   //-step-800---level--0-------------------------------------------------------------                                                 
   //            RE: crystal cool down without Ar
   //---------------------------------------------------------------------------------                                                 
           800 :                                                     
               IF #next_step[0] = #active_step[0] THEN                       
                   "APC".TI[0]       := 0;                     
                   "APC".OP_MSG      := "OP_MSG".RE_WAIT_TILL_XT_COOL;
                   "LT".AUTO_OP_CALL := FALSE;
                END_IF;

               // calculate all setpoints for this step
               // -------------------------------------                                      
               "AM_PAR_FNC_RE"();

               //argon inlet 
               //-----------
               "DC".V5_OP    := FALSE;   //close valve V5
               "DC".V6_OP    := TRUE;    //open valve V6

               //stop crystal rotation
               //---------------------
               IF ("DC".XT_ROT_CW OR "DC".XT_ROT_CCW) THEN 
                   IF "SysTick1s" THEN
                       "AC".SET_XT_ROT := "AC".SET_XT_ROT - ("CNF".RE_RMP_RTE_XT_ROT / 60.0);
                   END_IF;
               END_IF;

               IF ("AC".SET_XT_ROT <= 1.0)  THEN
                   "AC".SET_XT_ROT   :=  0.0;
                   "DC".XT_ROT_CW    :=  FALSE;
                   "DC".XT_ROT_CCW   :=  FALSE;
               END_IF;

               // time till end of this step
               // --------------------------
               "APC".ACT_TME_STE := (REAL_TO_INT("PAR_MAIN".RC_XT_COOL_DN_TME) * 60) - "APC".TI[0];

               //check end condition
               //-------------------
               IF (("APC".TI[0] > (REAL_TO_INT("PAR_MAIN".RC_XT_COOL_DN_TME) * 60)) AND ("AC".SET_XT_ROT = 0.0)) THEN    
                   #end_of_step[0] := true;                            
               END_IF;

               #next_step[0] := 900; 

   //-step-900---level--0-------------------------------------------------------------                                                 
   //            RE: increase pressure in gate chamber
   //---------------------------------------------------------------------------------                                                 
           900 :                                                     
               IF #next_step[0] = #active_step[0] THEN
                   "APC".OP_MSG := "OP_MSG".VENTING_GATE;
               END_IF;

               // calculate all setpoints for this step
               // -------------------------------------                                      
               "AM_PAR_FNC_RE"();

               //vent gate chamber
               //-----------------
               IF  ("LT".V7_CLOSE AND NOT "LT".V7_OPEN)  THEN  // gate valve V7 closed ?
                   "DC".V4_OP            := TRUE;
                   "FLT".GATE_V_NOT_CLD  := FALSE;
               ELSE
                   "DC".V4_OP            := FALSE;
                   "FLT".GATE_V_NOT_CLD  := TRUE;
               END_IF;

               //check end condition
               //-------------------
               IF "DV".APS_GCH_DELAYED THEN    
                   "DC".V4_OP        := FALSE;
                   #end_of_step[0]  := true;                            
               END_IF;

               #next_step[0] := 1000; 

   //-step-1000---level--0------------------------------------------------------------                                                 
   //            RE: crystal cool down with Ar and raise crucible to start position
   //---------------------------------------------------------------------------------                                                 
          1000 :                                                     
               IF #next_step[0] = #active_step[0] THEN                       
                   "APC".TI[0]   := 0;                     
                   "APC".OP_MSG  := "OP_MSG".RE_WAIT_TILL_XT_COOL;
                END_IF;

               // calculate all setpoints for this step
               // -------------------------------------                                      
               "AM_PAR_FNC_RE"();

               // time till end of this step
               // --------------------------
               "APC".ACT_TME_STE := (REAL_TO_INT("PAR_MAIN".RC_XT_COOL_DN_TME_AR) * 60) - "APC".TI[0];

               //raise crucible to start position
               //--------------------------------
               IF ("AV".ACT_CR_POS < #cr_start_pos) THEN
                   "DC".CR_LFT_UP    :=  TRUE;    
                   "AC".SET_CR_SPD   :=  "CNF".RE_CR_SPD;
               ELSE
                   IF NOT "APC".AUTOMATIC THEN                       //stop crucible lift if puller running in manual mode
                       IF "DC".CR_LFT_UP THEN
                           "KYD".CR_LFT_OFF  :=  TRUE;
                           #cr_lft_man_off  :=  true;
                       ELSIF #cr_lft_man_off THEN 
                           "KYD".CR_LFT_OFF  :=  FALSE;
                           #cr_lft_man_off  :=  false;
                       END_IF;
                   END_IF;
                   "DC".CR_LFT_UP    :=  FALSE;    
                   "AC".SET_CR_SPD   :=  0.0;
               END_IF;

               //check end condition
               //-------------------
               IF (("APC".TI[0] > (REAL_TO_INT("PAR_MAIN".RC_XT_COOL_DN_TME_AR) * 60)) AND NOT "DC".CR_LFT_UP) THEN    
                   #end_of_step[0] := true;                            
               END_IF;

               #next_step[0] := 1050; 

   //-step-1050--level--0---------------------------------------------------------------------------------------------                                                
   //            RE: check if gate chamber is at atmospheric pressure
   //-----------------------------------------------------------------------------------------------------------------                                   
           1050 :                                                     
               IF #next_step[0] = #active_step[0] THEN                       
                   "APC".TI[0]   := 0;                     
               END_IF;

               // calculate all setpoints for this step
               // -------------------------------------                                      
               "AM_PAR_FNC_RE"();

               //check end condition
               //-------------------
               IF "DV".APS_GCH_DELAYED THEN    
                   "DC".V4_OP            := FALSE;
                   "FLT".GATE_V_NOT_CLD  := FALSE;
               ELSE
                   IF  ("LT".V7_CLOSE AND NOT "LT".V7_OPEN) THEN  // gate valve V7 closed ?
                       "DC".V4_OP            := TRUE;
                       "FLT".GATE_V_NOT_CLD  := FALSE;
                   ELSE
                       "DC".V4_OP            := FALSE;
                       "FLT".GATE_V_NOT_CLD  := TRUE;
                   END_IF;
               END_IF;

               //check end condition
               //-------------------
               IF (NOT "DC".V4_OP AND NOT "PDO".V4) THEN    
                   #end_of_step[0]  := true;                            
               END_IF;

               #next_step[0] := 1100; 

   //-step-1100--level--0---------------------------------------------------------------------------------------------                                                
   //            RE: message "remove crystal" and wait till crystal is removed  - increase crucible rot to start value
   //-----------------------------------------------------------------------------------------------------------------                                   
           1100 :                                                     
               IF #next_step[0] = #active_step[0] THEN                       
                   "APC".OP_MSG          :=  "OP_MSG".RE_REMOVE_CRYSTAL;
                   "LT".AUTO_OP_CALL     :=  TRUE;
                   "APC".TI[0]           :=  0;
                   #xt_removed          :=  false;
                   "KYD".CR_LFT_OFF      :=  FALSE;
                   "DV".MAN_ACKN_XT_RMV  :=  FALSE;
                   "LT".SHOW_XT_RMV_BTN  :=  TRUE;
               END_IF;

               // calculate all setpoints for this step
               // -------------------------------------                                      
               "AM_PAR_FNC_RE"();

               //crucible rotation set point ramp
               //--------------------------------
               IF ("SysTick1s" AND ("AC".SET_CR_ROT < #cr_start_rot)) THEN 
                   "AC".SET_CR_ROT := "AC".SET_CR_ROT + ("CNF".RE_RMP_RTE_CR_ROT / 60.0);
               END_IF;

               //built crystal removed flag
               //--------------------------
               IF NOT "PDI".LS_GCH_DOOR_CL AND "PDI".LS_GCH_DOOR_OP AND "PDI".LS_XT_HDL_SW_LOCK AND "PDI".LS_XT_SLID_FW AND "PDI".LS_UP_XT_CLP_CL THEN
                   #xt_removed := true;
               END_IF;

               //check end condition - crystal removed and puller closed again
               //-------------------------------------------------------------
               IF ("PDI".LS_GCH_DOOR_CL AND NOT "PDI".LS_GCH_DOOR_OP AND #xt_removed) OR "DV".MAN_ACKN_XT_RMV THEN 
                   //delay next step 5 seconds
                   //-------------------------
                   IF ("APC".TI[0] > 5) THEN    
                       IF ("AC".SET_CR_ROT >= #cr_start_rot) THEN  //crucible rot set point reached
                           #end_of_step[0] := true; 
                       END_IF;
                   END_IF;
               ELSE
                   "APC".TI[0] := 0;
               END_IF;

               #next_step[0] := 1200; 

   //-step-1200--level--0--------------------------------------------------------------                                                 
   //            RE: pump down gate chamber
   //----------------------------------------------------------------------------------                                                 
          1200 :                                                     
               IF #next_step[0] = #active_step[0] THEN
                   "APC".OP_MSG          := "OP_MSG".PUMP_DOWN_GATE;     
                   "LT".AUTO_OP_CALL     := FALSE;
                   "LT".SHOW_XT_RMV_BTN  := FALSE;
               END_IF;

               // calculate all setpoints 
               // -----------------------
               "AM_PAR_FNC_RE" ();

               //start vacuum pump
               //-----------------
               "DC".P3_ON := TRUE;

               //check if final pressure is reached
               //----------------------------------
               IF ("AV".ACT_PRS_GCH <= "PAR_MAIN".RC_PRG_STR_PRS)  THEN
                   "DC".V3_OP    := FALSE;  //close vacuum valve to gate chamber

               ELSE
                   "DC".V3_OP    := TRUE;   //open vacuum valve to gate chamber

               END_IF;

               //check end condition
               //-------------------
               IF NOT "PDO".V3 AND NOT "DC".V3_OP THEN     //vacuum valve V3 closed?
                   #end_of_step[0] := true;                            
               END_IF;

               #next_step[0] := 1300; 

   //-step-1300---level--0------------------------------------------------------------                                                 
   //            RE: purge Ar to furnace
   //---------------------------------------------------------------------------------                                                 
          1300 :                                                     
               IF #next_step[0] = #active_step[0] THEN
                   "APC".OP_MSG  := "OP_MSG".VENTING_GATE;       
                   "APC".TI[0]   :=  0;                                           
               END_IF;

               // calculate all setpoints 
               // -----------------------
               "AM_PAR_FNC_RE" ();

               // time till end of this step
               // --------------------------
               "APC".ACT_TME_STE := REAL_TO_INT("PAR_MAIN".RC_PRG_TME) - "APC".TI[0];

               //start purging
               //-------------
               IF (("APC".TI[0] <= REAL_TO_INT("PAR_MAIN".RC_PRG_TME)) AND NOT "PDI".GCH_APS)  THEN 
                   IF  ("LT".V7_CLOSE AND NOT "LT".V7_OPEN)THEN  // gate valve V7 closed ?
                       "DC".V4_OP            := TRUE;
                       "FLT".GATE_V_NOT_CLD  := FALSE;
                   ELSE
                       "DC".V4_OP            := FALSE;
                       "FLT".GATE_V_NOT_CLD  := TRUE;
                       "APC".TI[0]           := 0;
                   END_IF;
               //purging over
               //------------
               ELSE 
                   "DC".V4_OP            := FALSE;
                   "FLT".GATE_V_NOT_CLD  := FALSE;
                   #end_of_step[0]      := true;                            
               END_IF;

               #next_step[0] := 1400;   

   //-step-1400---level--0------------------------------------------------------------                                                 
   //            RE: check if additional purge cycle is requested
   //---------------------------------------------------------------------------------                                                 
          1400 :                                                     
               IF #next_step[0] = #active_step[0] THEN
                   "APC".OP_MSG  :=  "OP_MSG".BLANK;       
                   "APC".TI[0]   :=  0;            
                   #prg_cyc_cnt :=  #prg_cyc_cnt + 1;    //count amount of purge cycles                              
               END_IF;

               //delay switching to next step
               //----------------------------
               IF ("APC".TI[0] > 2) THEN
                   #end_of_step[0] := true;                            
               END_IF;

               //select next step
               //----------------
               IF (#prg_cyc_cnt >= REAL_TO_INT("PAR_MAIN".RC_AMT_PRG_CYC)) THEN
                   #next_step[0] := 1500; 
               ELSE
                   #next_step[0] := 1200; 
               END_IF;

   //-step-1500--level--0-------------------------------------------------------------                                                 
   //            RE: pump down gate chamber
   //---------------------------------------------------------------------------------                                                 
           1500 :                                                     
               IF #next_step[0] = #active_step[0] THEN                       
                   "APC".OP_MSG := "OP_MSG".PUMP_DOWN_GATE;
               END_IF;

               // calculate all setpoints for this step
               // -------------------------------------                                      
               "AM_PAR_FNC_RE"();

               //open vacuum valve to gate chamber
               //---------------------------------
               "DC".V3_OP    := TRUE;   

               //check end condition
               //-------------------
               IF ("AV".ACT_PRS_GCH < ("PAR_MAIN".RC_FIN_PRS_PMP_DN / 1000.0)) THEN        //unit of pressure is 10^-3 mbar
                   #end_of_step[0] := true;                            
               END_IF;

               #next_step[0] := 1600; 

   //-step-1600--level--0-------------------------------------------------------------                                                 
   //            RE: fill gate chamber with Argon
   //---------------------------------------------------------------------------------                                                 
           1600 :                                                     
               IF #next_step[0] = #active_step[0] THEN                       
                   "APC".OP_MSG := "OP_MSG".VENTING_GATE;
               END_IF;

               // calculate all setpoints for this step
               // -------------------------------------                                      
               "AM_PAR_FNC_RE"();

               //close vacuum valve to gate chamber
               //----------------------------------
               "DC".V3_OP    := FALSE;   

               //check end condition
               //-------------------
               IF (("AV".ACT_PRS_GCH - "CNF".RE_PRS_DIFF) < "AV".ACT_PRS_FCH) THEN    
                   IF  ("LT".V7_CLOSE AND NOT "LT".V7_OPEN) THEN  // gate valve V7 closed ?
                       "DC".V4_OP            := TRUE;
                       "FLT".GATE_V_NOT_CLD  := FALSE;
                   ELSE
                       "DC".V4_OP            := FALSE;
                       "FLT".GATE_V_NOT_CLD  := TRUE;
                   END_IF;
               ELSE      
                   "DC".V4_OP            := FALSE;
                   "FLT".GATE_V_NOT_CLD  := FALSE;
                   #end_of_step[0]      := true;                            
               END_IF;

               #next_step[0] := 1700; 

   //-step-1700--level--0-------------------------------------------------------------                                                 
   //            RE: message "open gate valve"
   //---------------------------------------------------------------------------------                                                 
           1700:                                                     
               IF #next_step[0] = #active_step[0] THEN                       
                   "APC".OP_MSG      := "OP_MSG".OPEN_GATE_VALVE;
                   "LT".AUTO_OP_CALL := TRUE;
               END_IF;

               // calculate all setpoints for this step
               // -------------------------------------                                      
               "AM_PAR_FNC_RE"();

               //switch off auxilliary pump
               //--------------------------
               "DC".P3_ON    :=  FALSE;  

               //open V5 when gate valve not closed
               //----------------------------------
               IF (NOT "LT".V7_CLOSE) THEN
                   "DC".V5_OP := TRUE;
               END_IF;

               //DC.V7_UP     := NOT PDI.LS_V7_UP;
               //DC.V7_SW_OUT := DV.LS_V7_UP_DLY AND NOT PDI.LS_V7_SW_OUT;

               //check end condition
               //-------------------
               IF (NOT "LT".V7_CLOSE AND "LT".V7_OPEN AND "DV".LS_V7_SW_OUT_DLY) THEN   //V7 open ?
                   "DC".V6_OP            := FALSE;               //close V6   
                   #end_of_step[0]      := true;                            
               END_IF;

               #next_step[0] := 1800; 

   //-step-1800--level--0-------------------------------------------------------------                                                 
   //            RE: wait for dipping (manual triggering of further action is necessary)
   //---------------------------------------------------------------------------------                                                 
           1800:                                                     
               "APC".OP_MSG      := "OP_MSG".RE_WAIT_FOR_DIP;
               "LT".AUTO_OP_CALL := FALSE;

               // calculate all setpoints for this step
               // -------------------------------------                                      
               "AM_PAR_FNC_RE"();

               #next_step[0] := 1800;                               // E N D

       END_CASE;

       #start_previous := #start;                                    //save start input for next call 
       #cont_previous := "APC".CONT;                                  //save cont input for next call 
       #resume_previous := "APC".RESUME;                              //save resume input for next call
       #jump_previous := "APC".JUMP;                                  //save jump input for next call
       #single_previous := "APC".SINGLE;                              //save single input for next call
END_FUNCTION_BLOCK

FUNCTION_BLOCK "AM_EMG"   // FB205, SCL
{ S7_Optimized_Access := 'FALSE' }
VERSION : 0.0
// --------------------------------------------------------------------------------
//     program     :    AM_EMG
//     description :    apc emergency module  
//     name        :    G. Eibelsh鋟ser
//     date        :    02.11.2004
// 
//     revision    :    
//     name        :    
//     date        :    
//                     (c)CGS
//     --------------------------------------------------------------------------------
   VAR_INPUT
      start : Bool;   // start sequence, activate step 10 (impulse triggered)
   END_VAR
   VAR
      start_previous : Bool;   // start input value of last call
      cont_previous : Bool;   // cont input value of last call
      resume_previous : Bool;   // resume input value of last call
      jump_previous : Bool;   // jump input value of last call
      single_previous : Bool;   // single input value of last call
      active_step : Array[0..7] of Int;   // active step number for sequence level 0..7
      next_step : Array[0..7] of Int;   // next step number for sequence level 0..7
      hold_step : Array[0..7] of Int;   // step number of step on hold
      end_of_step : Array[0..7] of Bool;   // active step is done flag for sequence 0..7
      EndOfStep : Bool;   // default value for active step is done flag
      cont_enable : Array[0..7] of Bool;   // enable continue function
      ContEnable : Bool;   // default value for enable continue function
      cr_in_pos : Bool;   // crucible in safe position
      xt_in_pos : Bool;   // crystal in safe position
      set_xt_pos : Real;   // setpoint crystal position
      set_cr_pos : Real;   // setpoint crucible position
      start_pos_xt : Real;
   END_VAR
BEGIN


       "APC".STATUS := "APC".EMG;                                      // set apc status               

       "AM_SEQUENCE_CTL" (start_p            := #start,               // control sequence
                        start_previous_p   := #start_previous,
                        cont_previous_p    := #cont_previous, 
                        resume_previous_p  := #resume_previous,
                        jump_previous_p    := #jump_previous,
                        single_previous_p  := #single_previous,
                        active_step_p      := #active_step, 
                        next_step_p        := #next_step,
                        hold_step_p        := #hold_step, 
                        end_of_step_p      := #end_of_step, 
                        cont_enable_p      := #cont_enable); 


       CASE #active_step[0] OF    //sequence level_0
   //step--0-----level--0-------------------------------------------------off--(sequence off)--------------
           0    :                                                  
                #next_step[0] := 0;

   //step--1-----level--0-------------------------------------------------hold-(test sequence)-------------
           1   :                                                       
               IF #next_step[0] = #active_step[0] THEN                   //init step     
                   //init code
                   ; 
               END_IF;
               //step code                                             //do step
               ;
   //-step-10----level--0----------------------------------------------main-(start sequence)---------------                                                 
   //-step-10----level--0-------------------------------------------------------------                                                 
   //            EMG: init emergency sequence
   //---------------------------------------------------------------------------------                                                 
           10  :  

               // enable automatic mode
               // ---------------------
               "DC".MOD_AUT_ENB  := TRUE;

               "DV".HOR_OPP  := FALSE;
               "DV".LMP_OR   := TRUE;

               #cr_in_pos   := FALSE;
               #xt_in_pos   := FALSE;

               // init rotation drives
               // --------------------
               "DC".XT_ROT_CW    := FALSE;       
               "DC".XT_ROT_CCW   := FALSE;     

               "DC".CR_ROT_CW    := FALSE;    
               "DC".CR_ROT_CCW   := FALSE;   

               "AC".SET_XT_SPD   := 0.0;
               "AC".SET_XT_ROT   := 0.0;
               "AC".SET_CR_SPD   := 0.0;
               "AC".SET_CR_ROT   := 0.0;

               // heater
               // ------
               "DC".HTR_1_ON     :=  FALSE;                    
               "DC".HTR_2_ON     :=  FALSE;

               //mobile feeder
               //-------------
               "DC".MOB_FDR_MVE_IN_SEQ_ON    :=  FALSE;
               IF ("LT".MOB_FDR_DCK_DONE AND ("DV".FDG_MVE_IN_SEQ_DONE OR NOT "DV".FDG_MVE_OUT_SEQ_DONE)) THEN 
                   "DC".MOB_FDR_MVE_OUT_SEQ_ON   :=  TRUE;
               ELSE
                   "DC".MOB_FDR_MVE_OUT_SEQ_ON   :=  FALSE;
               END_IF;

               "DC".MOB_FDR_VIB_ON           :=  FALSE;
               "FLT".MOB_FDR_NOT_DCK         :=  FALSE;
               "FLT".MOB_FDR_STP_PARA        :=  FALSE;

               // init measurement system
               // -----------------------
               "DC".CAM_ISP_ON   :=  FALSE;          //inspection off
               "DC".CAM_INIT     :=  FALSE;
               "DC".CAM_MLT      :=  FALSE;
               "DC".CAM_DIP      :=  FALSE;
               "DC".CAM_DIA      :=  TRUE;
               "DC".CAM_SEL_1    :=  TRUE;
               "DC".CAM_SEL_2    :=  FALSE;

               // control loops
               // -------------
               "DC".CTL_DIA_ON       := FALSE;              // all control loops off
               "DC".CTL_GRW_RTE_ON   := FALSE;
               "DC".CTL_PULL_RTE_ON  := FALSE;
               "DC".CTL_CRUC_ROT_ON  := FALSE;
               "DC".CTL_MLT_LVL_ON   := FALSE;
               "DC".CTL_MLT_1_TMP_ON := FALSE;
               "DC".CTL_MLT_2_TMP_ON := FALSE;
               "DC".CTL_MLT_DRIFT_ON := FALSE;
               "DC".CTL_GAP_ON       := FALSE;

               "DC".CTL_HTR_1_TMP_ON := FALSE;             // heater temp loop on
               "DC".CTL_HTR_2_TMP_ON := FALSE;

               "DC".CTL_PRS_ON        := TRUE;            // pressure control on

               "DC".CTL_SI_FDR_ON    := FALSE;
               "DC".CTL_DOP_FDR_ON   := FALSE;

               #end_of_step[0]  :=  true;
               #next_step[0] := 100;

   //-step-100---level--0-------------------------------------------------------------                                                 
   //            EMG: set control immediately to automatic mode
   //---------------------------------------------------------------------------------                                                 
           100 :                                                     

               "APC".AUTOMATIC       :=  TRUE;               
               "APC".ACT_TME_PROC    :=  0;          //reset phase time
               "APC".ACT_TME_STE     :=  0;          // reset time of step

               "APC".OP_MSG := "OP_MSG".BLANK;

               #end_of_step[0]  :=  true;                            
               #next_step[0]    :=  200;

   //-step-200---level--0-------------------------------------------------------------                                                 
   //            EMG: positioning of crystal and crucible
   //---------------------------------------------------------------------------------                                                 
           200 :   

               IF #next_step[0] = #active_step[0] THEN
                   //reset initial temperature and power setpoints
                   //----------------------------------------------
                   "DIS".HTR_1_TMP_SET_PHA_STR   :=  0.0;
                   "DIS".HTR_2_PWR_SET_PHA_STR   :=  0.0;

                   #start_pos_xt    :=  "AV".ACT_XT_POS;      //store actual crystal position                                                
               END_IF;

               //check limits of crucible movement
               //---------------------------------
               IF ("PAR_MAIN".MCONST_EMG_CR_POS < "PAR_MAIN".MCONST_LIM_CR_DN) THEN
                   #set_cr_pos := "PAR_MAIN".MCONST_LIM_CR_DN;
               ELSIF ("PAR_MAIN".MCONST_EMG_CR_POS > "PAR_MAIN".MCONST_LIM_CR_UP)  THEN
                   #set_cr_pos := "PAR_MAIN".MCONST_LIM_CR_UP;
               ELSE
                   #set_cr_pos := "PAR_MAIN".MCONST_EMG_CR_POS;       //set target position of crubible lift
               END_IF;

               "DC".CR_LFT_FST := TRUE;  //activate crucible fast flag

               //call crucible positioning module
               //--------------------------------
               "AM_CR_DRV_MOVE_DB"(set_pos   := #set_cr_pos,
                                               set_spd := "PAR_MAIN".MCONST_EMG_CR_SPD,
                                               act_pos := "AV".ACT_CR_POS, 
                                               cnf     := "CNF".CNF_CR_POS, 
                                               out_up  := "DC".CR_LFT_UP,
                                               out_dn  := "DC".CR_LFT_DN, 
                                               out_spd := "AC".SET_CR_SPD,
                                               done    := #cr_in_pos);

               //check upper limit of crystal movement
               //-------------------------------------
               IF ((#start_pos_xt - "PAR_MAIN".MCONST_EMG_XT_LFT_DIST) < "PAR_MAIN".MCONST_LIM_XTAL_UP) THEN
                   #set_xt_pos := "PAR_MAIN".MCONST_LIM_XTAL_UP;
               ELSE
                   #set_xt_pos := #start_pos_xt - "PAR_MAIN".MCONST_EMG_XT_LFT_DIST; //calculate target position crystal lift
               END_IF;

               //do lifting up of crystal
               //------------------------
               IF ("AV".ACT_XT_POS > #set_xt_pos) THEN
                   "DC".XT_LFT_UP    :=  TRUE;
                   "AC".SET_XT_SPD   :=  "PAR_MAIN".MCONST_EMG_XT_SPD;

                   IF ("AC".SET_XT_SPD > "CNF_XT_LFT_LZ950".MAX_SPEED)   THEN
                       "DC".XT_LFT_FST := TRUE;       
                   ELSE
                       "DC".XT_LFT_FST := FALSE;
                   END_IF;

               ELSE                            //stop drive, target position reached
                   "DC".XT_LFT_UP    :=  FALSE;
                   "DC".XT_LFT_FST   :=  FALSE;       
                   "AC".SET_XT_SPD   :=  0.0;           
                   #xt_in_pos       :=  true;
               END_IF;

               //check end condition
               //-------------------
               IF #cr_in_pos AND #xt_in_pos THEN
                   #end_of_step[0]  :=  true;
               END_IF;

               #next_step[0] := 300; 

   //-step-300---level--0-------------------------------------------------------------                                                 
   //            EMG: switch to manual and wait
   //---------------------------------------------------------------------------------                                                 
           300 : 

               // disable automatic mode
               // ----------------------
               "DC".MOD_AUT_ENB  := false;

               #next_step[0] := 300;

   //---------------------------------------------------------------------------------                                                 
       END_CASE;

       #start_previous  := #start;           //save start input for next call 
       #cont_previous   := "APC".CONT;        //save cont input for next call 
       #resume_previous := "APC".RESUME;      //save resume input for next call
       #jump_previous   := "APC".JUMP;        //save jump input for next call
       #single_previous := "APC".SINGLE;      //save single input for next call
END_FUNCTION_BLOCK

FUNCTION_BLOCK "AM_BY2_RP_CALC_INC"   // FB251, SCL
{ S7_Optimized_Access := 'FALSE' }
VERSION : 0.0
// --------------------------------------------------------------------------------
//     program     :    AM_BY2_RP_CALC_INC
//     description :    Calculate increment value/100ms for crystal length ramp for 2nd body
// 
//     name        :    M.Lech  
//     date        :    23.04.01
// 
//     revision    :    
//     name        :    
//     date        :    
//                     (c) CGS
//     --------------------------------------------------------------------------------
   VAR
      t : Real;   // t in sec
      INC : Real;   // INC in mm/100msec
      INC_SUM : Real;
   END_VAR
BEGIN

      IF "PAR_MAIN".BY2_RP_TME <> 0.0 THEN               //disable ramp if time = 0.0
       IF #t < "PAR_MAIN".BY2_RP_TME AND "AV".ACT_XT_LEN >= "PAR_MAIN".BY2_LEN_RP_START THEN    
           #INC := ("PAR_MAIN".BY_XT_LEN - "KYA".ACT_BDY2_LEN)/("PAR_MAIN".BY2_RP_TME*10);          // (Ltot-Lby2)/T; inc/100msec
           #INC_SUM := #INC_SUM + #INC;
           #t := #t + 0.1;                              // t+100msec     
           "APC".OP_MSG := "OP_MSG".BY2_RAMP_ACTIVE;
       ELSE    
           "APC".OP_MSG := "OP_MSG".BLANK;
       END_IF;
      END_IF;
END_FUNCTION_BLOCK

FUNCTION_BLOCK "AM_PRS_CTRL"   // FB252, SCL
{ S7_Optimized_Access := 'FALSE' }
VERSION : 0.0
// --------------------------------------------------------------------------------
//     program     :    AM_PRS_CTRL
//     description :    Controls pressure and gas flow.
// 
//                           gas flow setp > 0:    pressure control on
// 
//                                         = 0:    pressure control off
//                                                 V4 or V1 open till pressure
//                                                 setpoint reached
// 
// 
//     name        :    D.Bruess
//     date        :    19.11.99
// 
//     revision    :    
//     name        :    
//     date        :    
//                     (c) CGS
//     --------------------------------------------------------------------------------
   VAR_INPUT
      set_prs : Real;   // setpoint for pressure
      set_flw_1 : Real;   // setpoint for gas flow 1
      set_flw_2 : Real;   // setpoint for gas flow 2
      act_prs : Real;   // actual pressure
   END_VAR
   VAR_IN_OUT
      out_V4 : Bool;   // valve for venting
      out_V5 : Bool;   // valve for gas inlet
      out_prs_ctl : Bool;   // pressure control on
      out_flw_1 : Real;   // output gas flow 1
      out_flw_2 : Real;   // output gas flow 2
      out_prs : Real;   // output pressure setpoint
      out_valve_pos : Real;   // output throttle valve pos
      done : Bool;   // done flag
   END_VAR
   VAR
      req_vac : Bool;   // request flag vacuum
      req_vent : Bool;   // request flag vent
   END_VAR
BEGIN


     #out_prs := #set_prs;

     IF ((#set_flw_1 > 0.0) OR (#set_flw_2 > 0.0)) THEN
       // pressure control on (with gas flow)
       // -----------------------------------
       #out_V4 := FALSE;
       #out_V5 := TRUE;
       #out_prs_ctl := TRUE;
       #out_flw_1 := #set_flw_1;
       #out_flw_2 := #set_flw_2;
       #req_vac := FALSE;
       #req_vent := FALSE;

       #done := TRUE;
     ELSE
       // pressure control off (no gas flow)
       // ----------------------------------
       IF (#done = TRUE) THEN
         // close all valves
         // ----------------
         #out_V4 := FALSE;
         #out_V5 := FALSE;
         #out_prs_ctl := FALSE;
         #out_flw_1 := 0.0;
         #out_flw_2 := 0.0;
         #out_valve_pos := 0.0;
         #req_vac := FALSE;
         #req_vent := FALSE;
       ELSE
         IF (#set_prs < #act_prs) THEN
           // actual pressure above setpoint
           // ------------------------------
           IF (#req_vent = TRUE) THEN
             #req_vac := FALSE;                    // done
             #req_vent := FALSE;
             #done := TRUE;
           ELSE
             #req_vac := TRUE;                     // vacuum
             #req_vent := FALSE;
           END_IF;

         ELSE;
           // actual pressure below setpoint
           // ------------------------------
           IF (#req_vac = TRUE) THEN
             #req_vac := FALSE;                    // done
             #req_vent := FALSE;
             #done := TRUE;
           ELSE
             #req_vac := FALSE;                    // venting
             #req_vent := TRUE;
           END_IF;
         END_IF;

         // pressure control off
         // --------------------
         #out_prs_ctl := FALSE;

         IF (#req_vac = TRUE) THEN
           // start vaccum
           // ------------
           #out_V4 := FALSE;
           #out_V5 := FALSE;
           #out_prs_ctl := FALSE;
           #out_flw_1 := 0.0;
           #out_flw_2 := 0.0;
           #out_valve_pos := 50.0;
         ELSE
           IF (#req_vent = TRUE) THEN
             // start venting
             // -------------
             #out_V4 := TRUE;
             #out_V5 := FALSE;
             #out_prs_ctl := FALSE;
             #out_flw_1 := 0.0;
             #out_flw_2 := 0.0;
             #out_valve_pos := 0.0;
           ELSE
             // done (no request)
             // -----------------
             #out_V4 := FALSE;
             #out_V5 := FALSE;
             #out_prs_ctl := FALSE;
             #out_flw_1 := 0.0;
             #out_flw_2 := 0.0;
             #out_valve_pos := 0.0;
           END_IF;
         END_IF;
       END_IF;
     END_IF;
END_FUNCTION_BLOCK

FUNCTION_BLOCK "AM_DRV_MOVE"   // FB253, SCL
{ S7_Optimized_Access := 'FALSE' }
VERSION : 0.0
// --------------------------------------------------------------------------------
//     program     :    AM_DRV_MOVE
//     description :    Automatic positioning function (crystal and crucible).
// 
//                             set_spd        set_pos
//                         --------------------------------------------------
//                         1)     0              x        stop
//                         2)    pos             0        up with const speed
//                         3)    neg             0        dn with const speed
//                         4)    <>0            >0        move to set_pos
// 
//                      When the drive moves to set_pos then set_spd is used as 
//                      speed setpoint. If the actual position is (set_pos +- delta)
//                      then the speed setpoint is reduced. "delta" is calculated
//                      from the setpoint for the speed and from some configuration
//                      data. When the drive is in position the done flag is set.
//                      The positioning is restarted when the done flag is reset.
// 
//     name        :    D.Bruess
//     date        :    04.11.99
// 
//     revision    :    
//     name        :    
//     date        :    
//                     (c) CGS
//     --------------------------------------------------------------------------------
   VAR_INPUT
      set_pos : Real;   // setpoint for new position (0...max)
      set_spd : Real;   // setpoint for speed (0...max)
      act_pos : Real;   // actual position
      cnf : Struct
         d0 : Real;   // distance for switching to red. speed
         td : Real;   // delay time
         t_ramp : Real;   // time to reduce speed from v_max to 0
         v_max : Real;   // max speed in fast mode
         v_low : Real;   // min value for reduced speed
      END_STRUCT;
   END_VAR
   VAR_IN_OUT
      out_up : Bool;   // direction of movement = up
      out_dn : Bool;   // direction of mevement = down
      out_spd : Real;   // calculated setpoint speed
      done : Bool;   // a) set_pos=0: drive moves with const speeed
   END_VAR
   VAR
      delta : Real;   // position range for reduced setpoint
      pos_req : Bool;   // positioning has been started
   END_VAR
   VAR_TEMP
      set_spd_abs : Real;   // positive value of setpoint
      set_spd_reduced : Real;   // reduced speed setpoint
   END_VAR
BEGIN


     // calculate setpoints for speed and reduced speed
     // -----------------------------------------------
     #set_spd_abs := ABS (#set_spd);
     IF (#set_spd_abs > #cnf.v_low) THEN
       #set_spd_reduced := #cnf.v_low;
     ELSE
       #set_spd_reduced := #set_spd_abs;
     END_IF;

     // calculate distance for reduced speed
     // ------------------------------------
     #delta := #cnf.d0 +
              #cnf.td * #set_spd_abs / 60.0 +
              0.5 * #cnf.t_ramp * #set_spd_abs * #set_spd_abs / (#cnf.v_max * 60.0); 


     IF (#set_spd = 0.0) THEN
       // stop drive
       // ----------
       #out_up := FALSE;
       #out_dn := FALSE;
       #out_spd := 0.0;
       #done := TRUE;

     ELSE
       IF (#set_pos = 0.0) THEN
         // move up/dn with const speed
         // ---------------------------
         IF (#set_spd > 0.0) THEN
           // move up
           // -------
           #out_up := TRUE;
           #out_dn := FALSE;
           #out_spd := #set_spd_abs;
           #done := TRUE;

         ELSE
           // move down
           // ---------
           #out_up := FALSE;
           #out_dn := TRUE;
           #out_spd := #set_spd_abs;
           #done := TRUE;

         END_IF;

       ELSE
         IF ((#set_pos = #act_pos) OR (#done)) THEN
           // stop drive
           // ----------
           #out_up := FALSE;
           #out_dn := FALSE;
           #out_spd := 0.0;
           #done := TRUE;

         ELSE
           IF ((#act_pos < (#set_pos - #delta)) AND (#delta < #set_pos)) THEN
             // fast up
             // -------
             #out_up := TRUE;
             #out_dn := FALSE;
             #out_spd := #set_spd_abs;
             #pos_req := TRUE;

           ELSE
             IF (#act_pos > (#set_pos + #delta)) THEN
               // fast down
               // ---------
               #out_up := FALSE;
               #out_dn := TRUE;
               #out_spd := #set_spd_abs;
               #pos_req := TRUE;

             ELSE
               IF (#act_pos < #set_pos) THEN
                 IF (#pos_req AND #out_dn) THEN
                   // stop drive
                   // ----------
                   #out_up := FALSE;
                   #out_dn := FALSE;
                   #out_spd := 0.0;
                   #done := TRUE;

                 ELSE
                   // move up (with reduced speed)
                   // ----------------------------
                   #out_up := TRUE;
                   #out_dn := FALSE;
                   #out_spd := #set_spd_reduced;
                   #pos_req := TRUE;

                 END_IF;

               ELSE
                 IF (#pos_req AND #out_up) THEN
                   // stop drive
                   // ----------
                   #out_up := FALSE;
                   #out_dn := FALSE;
                   #out_spd := 0.0;
                   #done := TRUE;

                 ELSE
                   // move down (with reduced speed)
                   // ------------------------------
                   #out_up := FALSE;
                   #out_dn := TRUE;
                   #out_spd := #set_spd_reduced;
                   #pos_req := TRUE;

                 END_IF;
               END_IF;
             END_IF;
           END_IF;
         END_IF;
       END_IF;
     END_IF;


     // reset flag when positioning done
     // --------------------------------
     IF (#done = TRUE) THEN
       #pos_req := FALSE;
     END_IF;
END_FUNCTION_BLOCK

FUNCTION_BLOCK "SM_FLT_SETP_DEV_PRC"   // FB260, SCL
{ S7_Optimized_Access := 'FALSE' }
VERSION : 0.0
// --------------------------------------------------------------------------------
//     program     :    SM_CALL_FLT_SETP_DEV_PRC
//     description :    Setpoint deviation processing
//                      Call module to check deviation and set alarm flag       
//     name        :    G. Eibelsh鋟ser
//     date        :    04.02.00
// 
//     revision    :    alarms for magnet current and resistance
//     name        :    M. Lech
//     date        :    03.11.00
//     
//     revision    :    
//     name        :
//     date        :   
//                     (c) CGS
//     --------------------------------------------------------------------------------
   VAR
      ACT_FLT_TME_GAS_1_FLW : Int;   // actual fault time gas flow 1
      ACT_FLT_TME_GAS_2_FLW : Int;   // actual fault time gas flow 2
      ACT_FLT_TME_PRS : Int;   // actual fault time pressure
      ACT_FLT_TME_HTR_1_PWR : Int;   // actual fault time heater 1 power
      ACT_FLT_TME_HTR_2_PWR : Int;   // actual fault time heater 2 power
      ACT_FLT_TME_MAG_1_CUR : Int;   // actual fault time magnet 1 current
      ACT_FLT_TME_MAG_2_CUR : Int;   // actual fault time magnet 2 current
      ACT_FLT_TME_DIA_NECK_MIN : Int;   // actual fault time neck diameter below limit
      ACT_FLT_TME_XT_GRO : Int;   // actual fault time crystal growth
      ACT_FLT_TME_XT_1_DIA : Int;   // actual fault time crystal 1 diameter
      ACT_FLT_TME_XT_2_DIA : Int;   // actual fault time crystal 2 diameter
      ACT_FLT_TME_PULL_SPD_NE : Int;   // actual fault time average pull speed neck
      ACT_FLT_TME_PULL_SPD_BY1 : Int;   // actual fault time average pull speed body part 1
      ACT_FLT_TME_PULL_SPD_BY2 : Int;   // actual fault time average pull speed body part 2
   END_VAR
   VAR_TEMP
      dev_flt_gas_1_flw : Bool;   // fault flag gas flow 1
      dev_flt_gas_2_flw : Bool;   // fault flag gas flow 2
      dev_flt_prs : Bool;   // fault flag pressure
      dev_flt_htr_1_pwr : Bool;   // fault flag heater 1 power
      dev_flt_htr_2_pwr : Bool;   // fault flag heater 2 power
      dev_flt_mag_1_cur : Bool;   // fault flag magnet 1 current
      dev_flt_mag_2_cur : Bool;   // fault flag magnet 2 current
      dev_flt_dia_neck_min : Bool;   // fault flag neck diameter below limit
      dev_flt_xt_gro : Bool;   // fault flag crystal growth
      dev_flt_xt_1_dia : Bool;   // fault flag crystal diameter part 1
      dev_flt_xt_2_dia : Bool;   // fault flag crystal diameter part 2
      dev_flt_avg_pull_spd_ne : Bool;   // fault flag average pull speed neck
      dev_flt_avg_pull_spd_by1 : Bool;   // fault flag average pull speed body part 1
      dev_flt_avg_pull_spd_by2 : Bool;   // fault flag average pull speed body part 2
   END_VAR
BEGIN

       //------------------------------------     
       //fault setpoint deviation: gas flow 1
       //------------------------------------    
       "SM_FLT_SETP_DEV_DLY" (act_value        := "DIS".ACT_GAS_1_FLW,       
                            set_value        := "DIS".SET_GAS_1_FLW,
                            max_dev          := "PAR_MAIN".LIM_GAS_1_FLW,
                            delay_time       := "PAR_MAIN".LIM_GAS_FLW_DLY,
                            enable           := ("PDO".V5 OR "PDO".V6), 
                            fault            => #dev_flt_gas_1_flw);

       "FLT".GAS_FLW_1_OUT_OF_RNG := "SysOndelay"
                                   (DIN     := #dev_flt_gas_1_flw,                     // fault input
                                    SetTime := REAL_TO_INT("PAR_MAIN".LIM_GAS_FLW_DLY), // delay time
                                    ActTime := #ACT_FLT_TME_GAS_1_FLW,                 // actual time value
                                    Tick    := "SysTick1s");                            // timebase (1s)

       //------------------------------------ 
       //fault setpoint deviation: gas flow 2
       //------------------------------------    
       "SM_FLT_SETP_DEV_DLY" (act_value        := "DIS".ACT_GAS_2_FLW,       
                            set_value        := "DIS".SET_GAS_2_FLW,
                            max_dev          := "PAR_MAIN".LIM_GAS_2_FLW,
                            delay_time       := "PAR_MAIN".LIM_GAS_FLW_DLY,
                            enable           := ("PDO".V5 OR "PDO".V6),
                            fault            => #dev_flt_gas_2_flw);

       "FLT".GAS_FLW_2_OUT_OF_RNG := "SysOndelay"
                                   (DIN     := #dev_flt_gas_2_flw,                     // fault input
                                    SetTime := REAL_TO_INT("PAR_MAIN".LIM_GAS_FLW_DLY), // delay time
                                    ActTime := #ACT_FLT_TME_GAS_2_FLW,                 // actual time value
                                    Tick    := "SysTick1s");                            // timebase (1s)

       //------------------------------------ 
       //fault setpoint deviation: pressure
       //------------------------------------    
       "SM_FLT_SETP_DEV_DLY" (act_value        := "DIS".ACT_PRS_CLF,       
                            set_value        := "DIS".SET_PRS_FNC,
                            max_dev          := "PAR_MAIN".LIM_PRS,
                            delay_time       := "PAR_MAIN".LIM_GAS_FLW_DLY,
                            enable           := "LT".CTL_PRS_ON,
                            fault            => #dev_flt_prs);

       "FLT".PRS_OUT_OF_RNG := "SysOndelay"
                             (DIN     := #dev_flt_prs,                              // fault input
                              SetTime := REAL_TO_INT("PAR_MAIN".LIM_GAS_FLW_DLY),    // delay time
                              ActTime := #ACT_FLT_TME_PRS,                          // actual time value
                              Tick    := "SysTick1s");                               // timebase (1s)

       //---------------------------------------- 
       //fault setpoint deviation: heater 1 power
       //----------------------------------------    
       "SM_FLT_SETP_DEV_DLY" (act_value        := "DIS".ACT_HTR_1_PWR,       
                            set_value        := "DIS".SET_HTR_1_PWR,
                            max_dev          := "PAR_MAIN".LIM_HTR_1_PWR,
                            delay_time       := "PAR_MAIN".LIM_HTR_PWR_DLY,
                            enable           := "LT".HTR_1_ON,
                            fault            => #dev_flt_htr_1_pwr);

       "FLT".HTR_1_PWR_OUT_OF_RNG := "SysOndelay"
                                   (DIN     := #dev_flt_htr_1_pwr,                        // fault input
                                    SetTime := REAL_TO_INT("PAR_MAIN".LIM_HTR_PWR_DLY),    // delay time
                                    ActTime := #ACT_FLT_TME_HTR_1_PWR,                    // actual time value
                                    Tick    := "SysTick1s");                               // timebase (1s)

       //---------------------------------------- 
       //fault setpoint deviation: heater 2 power
       //----------------------------------------    
       "SM_FLT_SETP_DEV_DLY" (act_value        := "DIS".ACT_HTR_2_PWR,       
                            set_value        := "DIS".SET_HTR_2_PWR,
                            max_dev          := "PAR_MAIN".LIM_HTR_2_PWR,
                            delay_time       := "PAR_MAIN".LIM_HTR_PWR_DLY,
                            enable           := "LT".HTR_2_ON,
                            fault            => #dev_flt_htr_2_pwr);

       "FLT".HTR_2_PWR_OUT_OF_RNG := "SysOndelay"
                                   (DIN     := #dev_flt_htr_2_pwr,                        // fault input
                                    SetTime := REAL_TO_INT("PAR_MAIN".LIM_HTR_PWR_DLY),    // delay time
                                    ActTime := #ACT_FLT_TME_HTR_2_PWR,                    // actual time value
                                    Tick    := "SysTick1s");                               // timebase (1s)

       //---------------------------------------------
       //fault setpoint deviation: heater 1 resistance
       //---------------------------------------------   
       IF ABS("AV".ACT_HTR_1_RES_CNG) > "PAR_MAIN".LIM_HTR_1_RES    THEN
           "FLT".HTR_1_RES_OUT_OF_RNG    :=    TRUE;
       ELSE    
           "FLT".HTR_1_RES_OUT_OF_RNG    :=    FALSE;
       END_IF;

       //---------------------------------------------
       //fault setpoint deviation: heater 2 resistance
       //---------------------------------------------    
       IF ABS("AV".ACT_HTR_2_RES_CNG) > "PAR_MAIN".LIM_HTR_2_RES    THEN
           "FLT".HTR_2_RES_OUT_OF_RNG    :=    TRUE;
       ELSE    
           "FLT".HTR_2_RES_OUT_OF_RNG    :=    FALSE;
       END_IF;

       (*
       //-----------------------------------------------
       //fault setpoint deviation: magnet coil 1 current
       //-----------------------------------------------    
       SM_FLT_SETP_DEV_DLY (act_value        := DIS.ACT_MAG_1_CUR,       
                            set_value        := DIS.SET_MAG_1_CUR,
                            max_dev          := PAR_MAIN.LIM_MAG_1_CUR,
                            delay_time       := PAR_MAIN.LIM_MAG_DLY,
                            enable           := LT.MAG_ON,
                            fault            := dev_flt_mag_1_cur);

       FLT.MAG_1_CUR_OUT_OF_RNG := SysOndelay
                                   (DIN     := dev_flt_mag_1_cur,                        // fault input
                                    SetTime := REAL_TO_INT(PAR_MAIN.LIM_MAG_DLY),        // delay time
                                    ActTime := ACT_FLT_TME_MAG_1_CUR,                    // actual time value
                                    Tick    := SysTick1s);                               // timebase (1s)

       //-----------------------------------------------
       //fault setpoint deviation: magnet coil 2 current
       //-----------------------------------------------    
       SM_FLT_SETP_DEV_DLY (act_value        := DIS.ACT_MAG_2_CUR,       
                            set_value        := DIS.SET_MAG_2_CUR,
                            max_dev          := PAR_MAIN.LIM_MAG_2_CUR,
                            delay_time       := PAR_MAIN.LIM_MAG_DLY,
                            enable           := LT.MAG_ON,
                            fault            := dev_flt_mag_2_cur);

       FLT.MAG_2_CUR_OUT_OF_RNG := SysOndelay
                                   (DIN     := dev_flt_mag_2_cur,                        // fault input
                                    SetTime := REAL_TO_INT(PAR_MAIN.LIM_MAG_DLY),        // delay time
                                    ActTime := ACT_FLT_TME_MAG_2_CUR,                    // actual time value
                                    Tick    := SysTick1s);                               // timebase (1s)


       //--------------------------------------------------
       //fault setpoint deviation: magnet coil 1 resistance
       //--------------------------------------------------   
       IF ABS(AV.ACT_MAG_1_RES_CNG) > PAR_MAIN.LIM_MAG_1_RES    THEN
           FLT.MAG_1_RES_OUT_OF_RNG    :=    TRUE;
       ELSE    
           FLT.MAG_1_RES_OUT_OF_RNG    :=    FALSE;
       END_IF;


       //--------------------------------------------------
       //fault setpoint deviation: magnet coil 2 resistance
       //--------------------------------------------------   
       IF ABS(AV.ACT_MAG_2_RES_CNG) > PAR_MAIN.LIM_MAG_2_RES    THEN
           FLT.MAG_2_RES_OUT_OF_RNG    :=    TRUE;
       ELSE    
           FLT.MAG_2_RES_OUT_OF_RNG    :=    FALSE;
       END_IF;
       *)
       //------------------------------------------------------
       //fault setpoint deviation: neck diameter below limit
       //------------------------------------------------------    
       (*
       SM_FLT_SETP_DEV_DLY (act_value        := DIS.ACT_XT_DIA,       
                            set_value        := DIS.SET_XT_DIA,
                            max_dev          := PAR_MAIN.LIM_DIA_NECK_MIN,
                            delay_time       := PAR_MAIN.LIM_DIA_NECK_DLY,
                            enable           := (APC.STATUS = APC.NECK) AND DC.CTL_DIA_ON AND LT.XT_LFT_UP,
                            fault            := dev_flt_dia_neck_min);
       *)
       IF ("APC".STATUS = "APC".NECK) AND "DC".CTL_DIA_ON AND "LT".XT_LFT_UP   THEN 
           IF ("DIS".ACT_XT_DIA < "PAR_MAIN".LIM_DIA_NECK_MIN) THEN
               #dev_flt_dia_neck_min := true;
           ELSE 
               #dev_flt_dia_neck_min := false;
           END_IF;
       ELSE
           #dev_flt_dia_neck_min := false;
       END_IF;

       "FLT".NECK_DIA_BELOW_LIMIT := "SysOndelay"
                                   (DIN     := #dev_flt_dia_neck_min,                   // fault input
                                    SetTime := REAL_TO_INT("PAR_MAIN".LIM_DIA_NECK_DLY), // delay time
                                    ActTime := #ACT_FLT_TME_DIA_NECK_MIN,               // actual time value
                                    Tick    := "SysTick1s");                             // timebase (1s)

       //----------------------------------------
       //fault setpoint deviation: crystal growth
       //----------------------------------------
       "SM_FLT_SETP_DEV_DLY" (act_value        := "DIS".ACT_XTAL_GRO,       
                            set_value        := "DIS".SET_XTAL_GRO,
                            max_dev          := "PAR_MAIN".LIM_GRO,
                            delay_time       := "PAR_MAIN".LIM_GRO_DLY,
                            enable           := "DC".CTL_GRW_RTE_ON,
                            fault            => #dev_flt_xt_gro);

       "FLT".XT_GROWTH_OUT_OF_RNG := "SysOndelay"
                                   (DIN     := #dev_flt_xt_gro,                    // fault input
                                    SetTime := REAL_TO_INT("PAR_MAIN".LIM_GRO_DLY), // delay time
                                    ActTime := #ACT_FLT_TME_XT_GRO,                // actual time value
                                    Tick    := "SysTick1s");                        // timebase (1s)

       //--------------------------------------------------------
       //fault setpoint deviation: crystal diameter (body part 1)
       //--------------------------------------------------------
       IF ("APC".STATUS = "APC".BODY) AND ("DIS".ACT_XT_LEN_MM <= "PAR_MAIN".LIM_LEN_BODY1) THEN

        "SM_FLT_SETP_DEV_DLY" (act_value        := "DIS".ACT_XT_DIA,       
                             set_value        := "DIS".SET_XT_DIA,
                             max_dev          := "PAR_MAIN".LIM_DIA_BODY_1,
                             delay_time       := "PAR_MAIN".LIM_DIA_DLY,
                             enable           := "DC".CTL_DIA_ON AND "LT".XT_LFT_UP, 
                             fault            => #dev_flt_xt_1_dia);

        "FLT".XT_DIA_OUT_OF_RNG    := "SysOndelay"
                                   (DIN     := #dev_flt_xt_1_dia,                 // fault input
                                    SetTime := REAL_TO_INT("PAR_MAIN".LIM_DIA_DLY),  // delay time
                                    ActTime := #ACT_FLT_TME_XT_1_DIA,               // actual time value
                                    Tick    := "SysTick1s");                         // timebase (1s)

       //--------------------------------------------------------
       //fault setpoint deviation: crystal diameter (body part 2)
       //--------------------------------------------------------
       ELSIF ("APC".STATUS = "APC".BODY) AND ("DIS".ACT_XT_LEN_MM > "PAR_MAIN".LIM_LEN_BODY1) THEN

        "SM_FLT_SETP_DEV_DLY" (act_value        := "DIS".ACT_XT_DIA,       
                             set_value        := "DIS".SET_XT_DIA,
                             max_dev          := "PAR_MAIN".LIM_DIA_BODY_2,
                             delay_time       := "PAR_MAIN".LIM_DIA_DLY,
                             enable           := "DC".CTL_DIA_ON AND "LT".XT_LFT_UP, 
                             fault            => #dev_flt_xt_2_dia);

        "FLT".XT_DIA_OUT_OF_RNG    := "SysOndelay"
                                    (DIN     := #dev_flt_xt_2_dia,                   // fault input
                                     SetTime := REAL_TO_INT("PAR_MAIN".LIM_DIA_DLY),  // delay time
                                     ActTime := #ACT_FLT_TME_XT_2_DIA,               // actual time value
                                     Tick    := "SysTick1s");                         // timebase (1s)

       ELSE
           "FLT".XT_DIA_OUT_OF_RNG   :=  FALSE;    

       END_IF;

       //-------------------------------------------------
       //fault setpoint deviation: average pull speed neck
       //-------------------------------------------------
       IF ("APC".STATUS = "APC".NECK) THEN
        "SM_FLT_SETP_DEV_DLY" (act_value        := "DIS".ACT_XT_AV_SPD,       
                             set_value        := "DIS".SET_XT_AV_SPD,
                             max_dev          := "PAR_MAIN".LIM_AV_SPD_NE,
                             delay_time       := "PAR_MAIN".LIM_AV_SPD_DLY,
                             enable           := "DC".CTL_PULL_RTE_ON AND "LT".XT_LFT_UP,
                             fault            => #dev_flt_avg_pull_spd_ne);

        "FLT".AVG_PULL_SPD_OUT_OF_RNG:= "SysOndelay"
                                      (DIN     := #dev_flt_avg_pull_spd_ne,              // fault input
                                       SetTime := REAL_TO_INT("PAR_MAIN".LIM_AV_SPD_DLY), // delay time
                                       ActTime := #ACT_FLT_TME_PULL_SPD_NE,              // actual time value
                                       Tick    := "SysTick1s");                           // timebase (1s)

       //--------------------------------------------------------
       //fault setpoint deviation: average pull speed body part 1
       //--------------------------------------------------------
       ELSIF ("APC".STATUS = "APC".BODY) AND ("DIS".ACT_XT_LEN_MM <= "PAR_MAIN".LIM_LEN_BODY1) THEN

        "SM_FLT_SETP_DEV_DLY" (act_value       := "DIS".ACT_XT_AV_SPD,       
                            set_value        := "DIS".SET_XT_AV_SPD,
                            max_dev          := "PAR_MAIN".LIM_AV_SPD_BY1,
                            delay_time       := "PAR_MAIN".LIM_AV_SPD_DLY,
                            enable           := "DC".CTL_PULL_RTE_ON AND "LT".XT_LFT_UP,
                            fault            => #dev_flt_avg_pull_spd_by1);

         "FLT".AVG_PULL_SPD_OUT_OF_RNG:= "SysOndelay"
                                      (DIN     := #dev_flt_avg_pull_spd_by1,             // fault input
                                       SetTime := REAL_TO_INT("PAR_MAIN".LIM_AV_SPD_DLY), // delay time
                                       ActTime := #ACT_FLT_TME_PULL_SPD_BY1,             // actual time value
                                       Tick    := "SysTick1s");                           // timebase (1s)

       //--------------------------------------------------------
       //fault setpoint deviation: average pull speed body part 2
       //--------------------------------------------------------
       ELSIF ("APC".STATUS = "APC".BODY) AND ("DIS".ACT_XT_LEN_MM > "PAR_MAIN".LIM_LEN_BODY1) THEN

        "SM_FLT_SETP_DEV_DLY" (act_value        := "DIS".ACT_XT_AV_SPD,       
                             set_value        := "DIS".SET_XT_AV_SPD,
                             max_dev          := "PAR_MAIN".LIM_AV_SPD_BY2,
                             delay_time       := "PAR_MAIN".LIM_AV_SPD_DLY,
                             enable           := "DC".CTL_PULL_RTE_ON AND "LT".XT_LFT_UP,
                             fault            => #dev_flt_avg_pull_spd_by2);

        "FLT".AVG_PULL_SPD_OUT_OF_RNG:= "SysOndelay"
                                     (DIN     := #dev_flt_avg_pull_spd_by2,             // fault input
                                      SetTime := REAL_TO_INT("PAR_MAIN".LIM_AV_SPD_DLY), // delay time
                                      ActTime := #ACT_FLT_TME_PULL_SPD_BY2,             // actual time value
                                      Tick    := "SysTick1s");                           // timebase (1s)

       ELSE
           "FLT".AVG_PULL_SPD_OUT_OF_RNG :=  FALSE;

       END_IF;
END_FUNCTION_BLOCK

FUNCTION_BLOCK "BM_MCC"   // FB261, SCL
{ S7_Optimized_Access := 'FALSE' }
VERSION : 0.0
// --------------------------------------------------------------------------------
//     program     :    BM_MCC
//     description :    melt contact function block, test mode, fault setting, lights
//                          
//     name        :    G. Eibelshaeuser
//     date        :    14.02.2000
// 
//     revision    :
//     name        :
//     date        :    
//                     (c)CGS
// --------------------------------------------------------------------------------
   VAR
      mcc_enb : Bool;
      mcc_test : Bool;
      mcc_contact : Bool;
      mcc_on_tme_flag : Bool;
      mcc_off_tme_flag : Bool;
      mcc_detect_flag : Bool;
      mcc_xt_out_of_melt : Bool;
      mcc_on_tme : S5Time;
      mcc_off_tme : S5Time;
      mcc_detect : S5Time;
      mcc_flt_dly : S5Time;
   END_VAR
BEGIN


       //read peripherie input
       //---------------------
       #mcc_contact := "PDI".MCC_CONTACT_XT;

       //melt contact control enable
       //---------------------------
       IF ("APC".AUTOMATIC AND "DC".MCC_ON AND NOT #mcc_on_tme_flag) THEN
           #mcc_enb := TRUE;                                                                // mcc enable in automatic mode
       ELSIF (NOT "APC".AUTOMATIC AND ("KYD".MCC_ON  OR #mcc_enb) AND NOT "KYD".MCC_OFF) THEN     // mcc enable in manual mode
           #mcc_enb := TRUE;           
       ELSE    
           #mcc_enb := FALSE;                                                               // mcc disabled
       END_IF;

       //on time flag for melt contact control
       //-------------------------------------     
       #mcc_on_tme := S_ODT(T_NO:= "BM_MCC_ON_TME",                                           // Timer Symbol
                           S   := "DC".MCC_ON AND #mcc_detect_flag AND NOT #mcc_off_tme_flag,  // Start Condition
                           TV  := T#5s,                                                    // Time Setpoint 
                           Q   => #mcc_on_tme_flag); 

       //off time flag for melt contact control
       //--------------------------------------    
       #mcc_off_tme := S_ODT(   T_NO:= "BM_MCC_OFF_TME",                  // Timer Symbol
                               S   := #mcc_on_tme_flag AND "DC".MCC_ON,   // Start Condition
                               TV  := T#10s,                           // Time Setpoint 
                               Q   => #mcc_off_tme_flag);

       //melt contact control test mode
       //------------------------------
       IF ("APC".AUTOMATIC AND "DC".MCC_TST_ON)    THEN                                                // mcc test in automatic mode
           #mcc_test := TRUE;
       ELSIF (NOT "APC".AUTOMATIC AND ("KYD".MCC_TST_ON OR #mcc_test) AND NOT "KYD".MCC_TST_OFF)  THEN    // mcc test in manual mode
           #mcc_test := TRUE;
       ELSE    
           #mcc_test := FALSE;                                                                      // mcc test disabled
       END_IF;

       //crystal out of melt alarm
       //-------------------------
       IF (("APC".STATUS = "APC".DIPPING) OR ("APC".STATUS = "APC".REMOVAL)) THEN
           #mcc_xt_out_of_melt  := FALSE;
       ELSIF (#mcc_enb AND NOT #mcc_detect_flag) THEN
           #mcc_xt_out_of_melt  := TRUE;
       ELSE    
           #mcc_xt_out_of_melt  := FALSE;
       END_IF;

       #mcc_flt_dly := S_ODT(   T_NO:= "FLT_OUT_OF_MELT_DLY",                             // Timer Symbol
                               S   := #mcc_xt_out_of_melt AND NOT "LT".MLT_GAP_SEARCH,    // Start Condition
                               TV  := T#5s,                                            // Time Setpoint 
                               Q   => "FLT".EC_XT_OUT_OF_MELT);                          // Set alarm xtal out of melt

       //melt contact control detection flag
       //-----------------------------------
       #mcc_detect := S_OFFDT(  T_NO:= "MELT_CON_DETECT_DLY",             // Timer Symbol
                               S   := ("DC".MCC_ON AND NOT #mcc_enb) OR   // melt contact control requested, but not in check cycle
                                       #mcc_contact,                    // xtal is in melt
                               TV  :=  T#3s,                           // Time Setpoint 
                               Q   =>  #mcc_detect_flag);               // delay flag xtal in melt

       "DV".DI_MCC_CONTACT := #mcc_detect_flag;

       //set light variables on PC screen
       //--------------------------------
       "LT".MCC_ON             := #mcc_enb OR ("APC".AUTOMATIC AND "DC".MCC_ON);
       "LT".MCC_TST_ON         := #mcc_test;
       "LT".XT_MELT_CONTACT    := #mcc_detect_flag;        // 1: Melt contact, 0: No melt contact

       // write peripherie output
       //------------------------ 
       "PDO".MCC_ENB_XT  := #mcc_enb;
       "PDO".MCC_TEST_XT := #mcc_test;
END_FUNCTION_BLOCK

FUNCTION_BLOCK "BM_XT_WGT_CALC"   // FB262, SCL
{ S7_Optimized_Access := 'FALSE' }
VERSION : 0.0
// --------------------------------------------------------------------------------
//     program     :    BM_XT_WEIGHT_CALC
//     description :    calculate crystal weight in SHOULDER and BODY for 
//                      display variable     
//     name        :    G. Eibelsh鋟ser
//     date        :    22.02.2000
// 
//     revision    :    calculation after fixed pulling length change
//                      reset variable inserted
//     name        :    G. Eibelsh鋟ser
//     date        :    27.03.2006
//     
//                     (c)CGS
// --------------------------------------------------------------------------------
   VAR
      xt_pos_old : Real;
      pull_lgh_inc : Real;
      xt_wgt_inc : Real;
   END_VAR
   VAR CONSTANT
      min_pull_lgh : Real := 0.5;   // minimum pulling length between two calculation cycles in mm
   END_VAR
BEGIN


       //reset crystal weight
       //--------------------
       IF  ("APC".STATUS = "APC".PUMP_DOWN)    OR      //phase pump down active 
           ("APC".STATUS = "APC".MELTING)      OR      //phase melting active
           ("APC".STATUS = "APC".DIPPING)      OR      //phase dipping active
           ("APC".STATUS = "APC".NECK)         THEN    //phase neck active

           "AV".ACT_XT_WGT_CALC  := 0.0;
           #xt_pos_old          := "AV".ACT_XT_POS;

       //calculate crystal weight
       //------------------------
       ELSIF  ("APC".STATUS = "APC".SHOULDER) OR       //phase shoulder active
               ("APC".STATUS = "APC".BODY)     THEN    //phase body active

           //check pulling length change 
           //---------------------------
           IF ((#xt_pos_old - "AV".ACT_XT_POS) >= #min_pull_lgh) THEN

               //calculate pulling length of last calc cycle
               //-------------------------------------------
               #pull_lgh_inc    := #xt_pos_old - "AV".ACT_XT_POS;

               //store actual crystal position of this calculation cycle
               //-------------------------------------------------------
               #xt_pos_old      := "AV".ACT_XT_POS;

               //calculation of weight increment in kg
               //-------------------------------------
               #xt_wgt_inc := #pull_lgh_inc * SQR("AV".ACT_XT_DIA) * "CNF".RHO_SOL_SI_ROOM * "CNF".PI / 4;

               //calculation of weight sum in kg
               //-------------------------------
               "AV".ACT_XT_WGT_CALC := "AV".ACT_XT_WGT_CALC + #xt_wgt_inc;

           END_IF;
       END_IF;

       //display actual calculated crystal weight
       //----------------------------------------
       "DIS".ACT_XT_WGT_CALC :=  "AV".ACT_XT_WGT_CALC;
END_FUNCTION_BLOCK

FUNCTION_BLOCK "BM_OP_CALL"   // FB340, SCL
{ S7_Optimized_Access := 'FALSE' }
VERSION : 0.0
// --------------------------------------------------------------------------------
//     program     :    BM_OP_CALL
//     description :    start horn and lamp to call operator after time x
//     name        :    M.Lech
//     date        :    14.06.00
// 
//     revision    :
//     name        :
//     date        :    
//                     (c)CGS
//     --------------------------------------------------------------------------------
   VAR
      ACT_OP_CALL_TME : Int;   // actual Time
      OP_CALL_ALM : Bool;   // flag for operator call on 1Hz cycle
   END_VAR
BEGIN


       "LT".OP_CALL_ON := ("LT".OP_CALL_ON OR "KYD".OP_CALL_ON) AND NOT 
                       ("KYD".OP_CALL_OFF);

       IF "KYD".OP_CALL_ACK THEN
           #ACT_OP_CALL_TME := 0;
       END_IF;

       "LT".OP_CALL_ALM:= "SysOndelay"(DIN     := "LT".OP_CALL_ON,                    //  operator call activated
                                   SetTime := REAL_TO_INT("KYA".SET_OP_CALL_TME), // delay time
                                   ActTime := #ACT_OP_CALL_TME,                  // actual time value
                                   Tick    := "SysTick1s");                       // timebase (1s);


       IF "SysTick2s" AND  "LT".OP_CALL_ALM AND NOT #OP_CALL_ALM THEN
           #OP_CALL_ALM := TRUE;                                        //call flag on 2s cycle
       ELSIF  "SysTick200ms" AND  "LT".OP_CALL_ALM AND #OP_CALL_ALM THEN
           #OP_CALL_ALM := FALSE;
       ELSIF  NOT  "LT".OP_CALL_ALM OR NOT "LT".OP_CALL_ON   THEN       
           #OP_CALL_ALM := FALSE;
       END_IF;       

       IF "LT".OP_CALL_ALM = TRUE THEN
           "APC".OP_MSG := "OP_MSG".OP_CALL_ALM;
       END_IF;
END_FUNCTION_BLOCK

FUNCTION_BLOCK "PM_MDI"   // FB400, SCL
{ S7_Optimized_Access := 'FALSE' }
VERSION : 0.0
// --------------------------------------------------------------------------------
//     program:         PM_MDI
//     description :    automatically generated PM_MDI
//     name:            hp
//     date        :    03.02.2021
// 
//     revision:
//     name:
//     Date:
//                     (c)CGS
//     --------------------------------------------------------------------------------
   VAR
      y : Bool;
      count : Int := 8;
   END_VAR
   VAR_TEMP
      x : Bool;
   END_VAR
BEGIN


       "MDI".CB_FLT_DC24V_K2 := "PDI".CB_FLT_DC24V_K2;
       "MDI".CB_FLT_AC400V_K2 := "PDI".CB_FLT_AC400V_K2;
       "MDI".SPARE_16_2 := "PDI".SPARE_16_2;
       "MDI".CB_FLT_AC230V := "PDI".CB_FLT_AC230V;
       "MDI".SPARE_16_4 := "PDI".SPARE_16_4;
       "MDI".SPARE_16_5 := "PDI".SPARE_16_5;
       "MDI".SPARE_16_6 := "PDI".SPARE_16_6;
       "MDI".SPARE_16_7 := "PDI".SPARE_16_7;
       "MDI".SPARE_17_0 := "PDI".SPARE_17_0;
       "MDI".UPS_24V_ALM := "PDI".UPS_24V_ALM;
       "MDI".UPS_24V_NRM := "PDI".UPS_24V_NRM;
       "MDI".EMO := "PDI".EMO;
       "MDI".EMS := "PDI".EMS;
       "MDI".SPARE_17_5 := "PDI".SPARE_17_5;
       "MDI".SPARE_17_6 := "PDI".SPARE_17_6;
       "MDI".SPARE_17_7 := "PDI".SPARE_17_7;
       "MDI".P1_WRN := "PDI".P1_WRN;
       "MDI".P1_FLT := "PDI".P1_FLT;
       "MDI".P1_IS_ON := "PDI".P1_IS_ON;
       "MDI".P1_WD := "PDI".P1_WD;
       "MDI".FIL_APS := "PDI".FIL_APS;
       "MDI".MON_TMP_P2 := "PDI".MON_TMP_P2;
       "MDI".MON_TMP_P1 := "PDI".MON_TMP_P1;
       "MDI".SPARE_18_7 := "PDI".SPARE_18_7;
       "MDI".FCH_LFT_SDL_NUT := "PDI".FCH_LFT_SDL_NUT;
       "MDI".LS_FCH_LFT_DN := "PDI".LS_FCH_LFT_DN;
       "MDI".LS_FCH_HOOK_WORK := "PDI".LS_FCH_HOOK_WORK;
       "MDI".LS_FCH_HOOK_HOME := "PDI".LS_FCH_HOOK_HOME;
       "MDI".LS_TEC_FLG_DN := "PDI".LS_TEC_FLG_DN;
       "MDI".TEC_FLG_SDL_NUT := "PDI".TEC_FLG_SDL_NUT;
       "MDI".LS_V11_COV_OP := "PDI".LS_V11_COV_OP;
       "MDI".LS_V11_COV_CL := "PDI".LS_V11_COV_CL;
       "MDI".GCH_APS := "PDI".GCH_APS;
       "MDI".FCH_APS := "PDI".FCH_APS;
       "MDI".FDR_APS := "PDI".FDR_APS;
       "MDI".FIL_2_APS := "PDI".FIL_2_APS;
       "MDI".SPARE_33_4 := "PDI".SPARE_33_4;
       "MDI".SPARE_33_5 := "PDI".SPARE_33_5;
       "MDI".LS_V2_1_OP := "PDI".LS_V2_1_OP;
       "MDI".LS_V2_1_CL := "PDI".LS_V2_1_CL;
       "MDI".CB_FLT_AC400V_K5 := "PDI".CB_FLT_AC400V_K5;
       "MDI".CB_FLT_DC24V_K5 := "PDI".CB_FLT_DC24V_K5;
       "MDI".LS_MAG_LFT_UP := "PDI".LS_MAG_LFT_UP;
       "MDI".LS_MAG_LFT_DN := "PDI".LS_MAG_LFT_DN;
       "MDI".SLS_MAG_LFT := "PDI".SLS_MAG_LFT;
       "MDI".MAG_LFT_SDL_NUT1 := "PDI".MAG_LFT_SDL_NUT1;
       "MDI".MAG_LFT_SDL_NUT2 := "PDI".MAG_LFT_SDL_NUT2;
       "MDI".MAG_LFT_SDL_NUT3 := "PDI".MAG_LFT_SDL_NUT3;
       "MDI".OIL_LVL_CR_SFT := "PDI".OIL_LVL_CR_SFT;
       "MDI".LS_V1_OP := "PDI".LS_V1_OP;
       "MDI".LS_V1_CL := "PDI".LS_V1_CL;
       "MDI".MP_ENB_K5 := "PDI".MP_ENB_K5;
       "MDI".SLS_TEC_FLG_LFT := "PDI".SLS_TEC_FLG_LFT;
       "MDI".SLS_FCH_LFT := "PDI".SLS_FCH_LFT;
       "MDI".COMP_AIR_OK := "PDI".COMP_AIR_OK;
       "MDI".COMP_AIR_2_OK := "PDI".COMP_AIR_2_OK;
       "MDI".LS_V1_1_CL := "PDI".LS_V1_1_CL;
       "MDI".LS_V1_1_OP := "PDI".LS_V1_1_OP;
       "MDI".LS_V3_4_OP := "PDI".LS_V3_4_OP;
       "MDI".LS_V3_4_CL := "PDI".LS_V3_4_CL;
       "MDI".LS_V3_3_OP := "PDI".LS_V3_3_OP;
       "MDI".LS_V3_3_CL := "PDI".LS_V3_3_CL;
       "MDI".LS_V2_11_OP := "PDI".LS_V2_11_OP;
       "MDI".LS_V2_11_CL := "PDI".LS_V2_11_CL;
       "MDI".ACC_FCH_OV_PRS_1 := "PDI".ACC_FCH_OV_PRS_1;
       "MDI".ACC_FCH_OV_PRS_2 := "PDI".ACC_FCH_OV_PRS_2;
       "MDI".SPARE_48_2 := "PDI".SPARE_48_2;
       "MDI".ACC_WTR_FLW_OUT_OK := "PDI".ACC_WTR_FLW_OUT_OK;
       "MDI".ACC_WTR_FLW_IN_OK := "PDI".ACC_WTR_FLW_IN_OK;
       "MDI".ACC_WTR_TMP_OUT_OK := "PDI".ACC_WTR_TMP_OUT_OK;
       "MDI".OV_PRS_1_FLT := "PDI".OV_PRS_1_FLT;
       "MDI".OV_PRS_2_FLT := "PDI".OV_PRS_2_FLT;
       "MDI".ACC_SC_WTR_OK := "PDI".ACC_SC_WTR_OK;
       "MDI".ACC_SC_WTR_ATV := "PDI".ACC_SC_WTR_ATV;
       "MDI".ACC_SC_HTR_OK := "PDI".ACC_SC_HTR_OK;
       "MDI".ACC_SC_HTR_ATV := "PDI".ACC_SC_HTR_ATV;
       "MDI".ACC_KEY_RST := "PDI".ACC_KEY_RST;
       "MDI".ACC_CB_FLT_DC24V := "PDI".ACC_CB_FLT_DC24V;
       "MDI".ACC_UPS_24V_ALM := "PDI".ACC_UPS_24V_ALM;
       "MDI".ACC_UPS_24V_NRM := "PDI".ACC_UPS_24V_NRM;
       "MDI".DPH_RPT_DET_OK := "PDI".DPH_RPT_DET_OK;
       "MDI".ACC_CB_FLT_AC230V := "PDI".ACC_CB_FLT_AC230V;
       "MDI".SPARE_90_2 := "PDI".SPARE_90_2;
       "MDI".SPARE_90_3 := "PDI".SPARE_90_3;
       "MDI".SPARE_90_4 := "PDI".SPARE_90_4;
       "MDI".SPARE_90_5 := "PDI".SPARE_90_5;
       "MDI".SPARE_90_6 := "PDI".SPARE_90_6;
       "MDI".SPARE_90_7 := "PDI".SPARE_90_7;
       "MDI".FU_P2_RDY := "PDI".FU_P2_RDY;
       "MDI".SPARE_144_1 := "PDI".SPARE_144_1;
       "MDI".LS_GCH_UP := "PDI".LS_GCH_UP;
       "MDI".LS_GCH_DN := "PDI".LS_GCH_DN;
       "MDI".LS_GCH_SW_IN := "PDI".LS_GCH_SW_IN;
       "MDI".LS_GCH_SW_CLN := "PDI".LS_GCH_SW_CLN;
       "MDI".LS_GCH_SW_OUT := "PDI".LS_GCH_SW_OUT;
       "MDI".LS_GCH_SW_LOCK := "PDI".LS_GCH_SW_LOCK;
       "MDI".SLS_GCH_LFT := "PDI".SLS_GCH_LFT;
       "MDI".LS_TCH_UP := "PDI".LS_TCH_UP;
       "MDI".LS_TCH_DN := "PDI".LS_TCH_DN;
       "MDI".LS_TCH_SW_IN := "PDI".LS_TCH_SW_IN;
       "MDI".LS_TCH_SW_CLN := "PDI".LS_TCH_SW_CLN;
       "MDI".LS_TCH_SW_OUT := "PDI".LS_TCH_SW_OUT;
       "MDI".LS_TCH_SW_LOCK := "PDI".LS_TCH_SW_LOCK;
       "MDI".LS_TCH_TILT_0 := "PDI".LS_TCH_TILT_0;
       "MDI".LS_TCH_TILT_30 := "PDI".LS_TCH_TILT_30;
       "MDI".KEY_XT_LFT_SRV := "PDI".KEY_XT_LFT_SRV;
       "MDI".LS_V7_UP := "PDI".LS_V7_UP;
       "MDI".LS_V7_DN := "PDI".LS_V7_DN;
       "MDI".LS_V7_SW_IN := "PDI".LS_V7_SW_IN;
       "MDI".LS_V7_SW_OUT := "PDI".LS_V7_SW_OUT;
       "MDI".LS_V7_FLP_OP := "PDI".LS_V7_FLP_OP;
       "MDI".LS_V7_CLN_POS := "PDI".LS_V7_CLN_POS;
       "MDI".LS_GCH_BEL_UP := "PDI".LS_GCH_BEL_UP;
       "MDI".LS_GCH_BEL_DN := "PDI".LS_GCH_BEL_DN;
       "MDI".LS_XT_SLID_BW := "PDI".LS_XT_SLID_BW;
       "MDI".LS_XT_SLID_FW := "PDI".LS_XT_SLID_FW;
       "MDI".LS_XT_SLID_MID := "PDI".LS_XT_SLID_MID;
       "MDI".LS_XT_CLP_CON := "PDI".LS_XT_CLP_CON;
       "MDI".LS_XT_TILT_90 := "PDI".LS_XT_TILT_90;
       "MDI".LS_XT_TILT_75 := "PDI".LS_XT_TILT_75;
       "MDI".LS_UP_XT_CLP_FLT := "PDI".LS_UP_XT_CLP_FLT;
       "MDI".SPARE_275_7 := "PDI".SPARE_275_7;
       "MDI".LS_UP_XT_CLP_OP := "PDI".LS_UP_XT_CLP_OP;
       "MDI".LS_UP_XT_CLP_CL := "PDI".LS_UP_XT_CLP_CL;
       "MDI".LS_UP_XT_CLP_SAVE := "PDI".LS_UP_XT_CLP_SAVE;
       "MDI".LS_UP_XT_CLP_PLATE := "PDI".LS_UP_XT_CLP_PLATE;
       "MDI".LS_LO_XT_CLP_FLT := "PDI".LS_LO_XT_CLP_FLT;
       "MDI".LS_LO_XT_CLP_OP := "PDI".LS_LO_XT_CLP_OP;
       "MDI".LS_LO_XT_CLP_CL := "PDI".LS_LO_XT_CLP_CL;
       "MDI".LS_LO_XT_CLP_SAVE := "PDI".LS_LO_XT_CLP_SAVE;
       "MDI".LS_LO_XT_CLP_PLATE := "PDI".LS_LO_XT_CLP_PLATE;
       "MDI".LS_HOI_TOOL_INST := "PDI".LS_HOI_TOOL_INST;
       "MDI".XT_DRP_OUT_PRT_1_CL := "PDI".XT_DRP_OUT_PRT_1_CL;
       "MDI".XT_DRP_OUT_PRT_1_OP := "PDI".XT_DRP_OUT_PRT_1_OP;
       "MDI".XT_DRP_OUT_PRT_2_CL := "PDI".XT_DRP_OUT_PRT_2_CL;
       "MDI".XT_DRP_OUT_PRT_2_OP := "PDI".XT_DRP_OUT_PRT_2_OP;
       "MDI".CB_FLT_AC400V_K8 := "PDI".CB_FLT_AC400V_K8;
       "MDI".CB_FLT_DC24V_K8 := "PDI".CB_FLT_DC24V_K8;
       "MDI".XT_DRP_OUT_PRT_3_CL := "PDI".XT_DRP_OUT_PRT_3_CL;
       "MDI".XT_DRP_OUT_PRT_3_OP := "PDI".XT_DRP_OUT_PRT_3_OP;
       "MDI".XT_DRP_OUT_PRT_4_CL := "PDI".XT_DRP_OUT_PRT_4_CL;
       "MDI".XT_DRP_OUT_PRT_4_OP := "PDI".XT_DRP_OUT_PRT_4_OP;
       "MDI".LS_XT_HDL_SW_UNLOCK := "PDI".LS_XT_HDL_SW_UNLOCK;
       "MDI".LS_XT_HDL_SW_LOCK := "PDI".LS_XT_HDL_SW_LOCK;
       "MDI".LS_GCH_DOOR_OP := "PDI".LS_GCH_DOOR_OP;
       "MDI".LS_GCH_DOOR_CL := "PDI".LS_GCH_DOOR_CL;
       "MDI".MCC_CONTACT_XT := "PDI".MCC_CONTACT_XT;
       "MDI".OIL_LVL_XT_SFT := "PDI".OIL_LVL_XT_SFT;
       "MDI".LS_XT_SFT_SRV_POS := "PDI".LS_XT_SFT_SRV_POS;
       "MDI".LS_XT_TOP_POS := "PDI".LS_XT_TOP_POS;
       "MDI".SLS_TCH_LFT := "PDI".SLS_TCH_LFT;
       "MDI".XT_ROT_CAM_TRG := "PDI".XT_ROT_CAM_TRG;
       "MDI".MP_ENB_K8 := "PDI".MP_ENB_K8;
       "MDI".MP_ENB_K9 := "PDI".MP_ENB_K9;
       "MDI".LS_V3_OP := "PDI".LS_V3_OP;
       "MDI".LS_V3_CL := "PDI".LS_V3_CL;
       "MDI".FDR_LS_V3_2_OP := "PDI".FDR_LS_V3_2_OP;
       "MDI".FDR_LS_V3_2_CL := "PDI".FDR_LS_V3_2_CL;
       "MDI".LSR_SEN_OBJ_DET := "PDI".LSR_SEN_OBJ_DET;
       "MDI".SPARE_280_5 := "PDI".SPARE_280_5;
       "MDI".SPARE_280_6 := "PDI".SPARE_280_6;
       "MDI".SPARE_280_7 := "PDI".SPARE_280_7;
       "MDI".LS_V11_OP := "PDI".LS_V11_OP;
       "MDI".LS_V11_CL := "PDI".LS_V11_CL;
       "MDI".FDR_HOP_CON := "PDI".FDR_HOP_CON;
END_FUNCTION_BLOCK

FUNCTION_BLOCK "PM_MDO"   // FB401, SCL
{ S7_Optimized_Access := 'FALSE' }
VERSION : 0.0
// --------------------------------------------------------------------------------
//     program:         PM_MDO
//     description :    automatically generated PM_MDO
//     name:            hp
//     date        :    03.02.2021
// 
//     revision:
//     name:
//     Date:
//                     (c)CGS
//     --------------------------------------------------------------------------------
   VAR
      y : Bool;
      count : Int := 8;
   END_VAR
   VAR_TEMP
      x : Bool;
   END_VAR
BEGIN


       "MDO".HOR_OPP_K2 := "PDO".HOR_OPP_K2;
       "MDO".LMP_RD_K2 := "PDO".LMP_RD_K2;
       "MDO".LMP_YE_K2 := "PDO".LMP_YE_K2;
       "MDO".LMP_GN_K2 := "PDO".LMP_GN_K2;
       "MDO".LMP_BU_K2 := "PDO".LMP_BU_K2;
       "MDO".HOR_MAG_ACTIVE := "PDO".HOR_MAG_ACTIVE;
       "MDO".LMP_MAG_ACTIVE := "PDO".LMP_MAG_ACTIVE;
       "MDO".SPARE_16_7 := "PDO".SPARE_16_7;
       "MDO".P1_ON := "PDO".P1_ON;
       "MDO".P3_ON := "PDO".P3_ON;
       "MDO".P2_ON := "PDO".P2_ON;
       "MDO".P1_SEAL_GAS := "PDO".P1_SEAL_GAS;
       "MDO".P3_SEAL_GAS := "PDO".P3_SEAL_GAS;
       "MDO".HTR_PWR_ON := "PDO".HTR_PWR_ON;
       "MDO".V10 := "PDO".V10;
       "MDO".MON_TMP_P2_RES := "PDO".MON_TMP_P2_RES;
       "MDO".SPARE_18_0 := "PDO".SPARE_18_0;
       "MDO".SPARE_18_1 := "PDO".SPARE_18_1;
       "MDO".SPARE_18_2 := "PDO".SPARE_18_2;
       "MDO".SPARE_18_3 := "PDO".SPARE_18_3;
       "MDO".SPARE_18_4 := "PDO".SPARE_18_4;
       "MDO".SPARE_18_5 := "PDO".SPARE_18_5;
       "MDO".SPARE_18_6 := "PDO".SPARE_18_6;
       "MDO".SPARE_18_7 := "PDO".SPARE_18_7;
       "MDO".V1_OP := "PDO".V1_OP;
       "MDO".V1_CL := "PDO".V1_CL;
       "MDO".SPARE_32_2 := "PDO".SPARE_32_2;
       "MDO".SPARE_32_3 := "PDO".SPARE_32_3;
       "MDO".SPARE_32_4 := "PDO".SPARE_32_4;
       "MDO".CR_ROT_ENB := "PDO".CR_ROT_ENB;
       "MDO".CR_LFT_ENB := "PDO".CR_LFT_ENB;
       "MDO".FU_FCB_HDL_ON := "PDO".FU_FCB_HDL_ON;
       "MDO".TEC_FLG_LFT_ENB := "PDO".TEC_FLG_LFT_ENB;
       "MDO".FCH_LFT_ENB := "PDO".FCH_LFT_ENB;
       "MDO".MAG_LFT_UP := "PDO".MAG_LFT_UP;
       "MDO".MAG_LFT_DN := "PDO".MAG_LFT_DN;
       "MDO".BRK_MAG_LFT := "PDO".BRK_MAG_LFT;
       "MDO".SPARE_33_5 := "PDO".SPARE_33_5;
       "MDO".SPARE_33_6 := "PDO".SPARE_33_6;
       "MDO".SPARE_33_7 := "PDO".SPARE_33_7;
       "MDO".V1_1_OP := "PDO".V1_1_OP;
       "MDO".V1_1_CL := "PDO".V1_1_CL;
       "MDO".SPARE_34_2 := "PDO".SPARE_34_2;
       "MDO".SPARE_34_3 := "PDO".SPARE_34_3;
       "MDO".SPARE_34_4 := "PDO".SPARE_34_4;
       "MDO".SPARE_34_5 := "PDO".SPARE_34_5;
       "MDO".SPARE_34_6 := "PDO".SPARE_34_6;
       "MDO".SPARE_34_7 := "PDO".SPARE_34_7;
       "MDO".ACC_SC_HTR_STR := "PDO".ACC_SC_HTR_STR;
       "MDO".ACC_SC_HTR_RST := "PDO".ACC_SC_HTR_RST;
       "MDO".ACC_SC_WTR_STR := "PDO".ACC_SC_WTR_STR;
       "MDO".ACC_SC_WTR_RST := "PDO".ACC_SC_WTR_RST;
       "MDO".ACC_ALM_LT_1 := "PDO".ACC_ALM_LT_1;
       "MDO".ACC_ALM_SND_1 := "PDO".ACC_ALM_SND_1;
       "MDO".ACC_ALM_LT_2 := "PDO".ACC_ALM_LT_2;
       "MDO".ACC_ALM_SND_2 := "PDO".ACC_ALM_SND_2;
       "MDO".FCH_HOOK_HOME := "PDO".FCH_HOOK_HOME;
       "MDO".FCH_HOOK_WORK := "PDO".FCH_HOOK_WORK;
       "MDO".UP_FCH_SW_BRK := "PDO".UP_FCH_SW_BRK;
       "MDO".LO_FCH_SW_BRK := "PDO".LO_FCH_SW_BRK;
       "MDO".TEC_FLG_SW_BRK := "PDO".TEC_FLG_SW_BRK;
       "MDO".V25 := "PDO".V25;
       "MDO".V2_1 := "PDO".V2_1;
       "MDO".V21 := "PDO".V21;
       "MDO".V19 := "PDO".V19;
       "MDO".V20 := "PDO".V20;
       "MDO".V22 := "PDO".V22;
       "MDO".V9_2 := "PDO".V9_2;
       "MDO".V22_1 := "PDO".V22_1;
       "MDO".V3_4 := "PDO".V3_4;
       "MDO".V3_3 := "PDO".V3_3;
       "MDO".V2_11 := "PDO".V2_11;
       "MDO".P2_FU_ON := "PDO".P2_FU_ON;
       "MDO".P2_FU_RES := "PDO".P2_FU_RES;
       "MDO".V4 := "PDO".V4;
       "MDO".V5 := "PDO".V5;
       "MDO".V6 := "PDO".V6;
       "MDO".V3 := "PDO".V3;
       "MDO".V3_2 := "PDO".V3_2;
       "MDO".V24 := "PDO".V24;
       "MDO".XT_DRP_OUT_PRT_CL := "PDO".XT_DRP_OUT_PRT_CL;
       "MDO".XT_DRP_OUT_PRT_OP := "PDO".XT_DRP_OUT_PRT_OP;
       "MDO".TCH_SW_LOCK := "PDO".TCH_SW_LOCK;
       "MDO".TCH_SW_UNLOCK := "PDO".TCH_SW_UNLOCK;
       "MDO".GCH_SW_LOCK := "PDO".GCH_SW_LOCK;
       "MDO".GCH_SW_UNLOCK := "PDO".GCH_SW_UNLOCK;
       "MDO".XT_HDL_SW_LOCK := "PDO".XT_HDL_SW_LOCK;
       "MDO".XT_HDL_SW_UNLOCK := "PDO".XT_HDL_SW_UNLOCK;
       "MDO".FDR_V11_OP := "PDO".FDR_V11_OP;
       "MDO".FDR_V11_CL := "PDO".FDR_V11_CL;
       "MDO".FDR_V11_CVR_OP := "PDO".FDR_V11_CVR_OP;
       "MDO".FDR_V11_CVR_CL := "PDO".FDR_V11_CVR_CL;
       "MDO".SPARE_226_2 := "PDO".SPARE_226_2;
       "MDO".SPARE_226_3 := "PDO".SPARE_226_3;
       "MDO".SPARE_226_4 := "PDO".SPARE_226_4;
       "MDO".SPARE_226_5 := "PDO".SPARE_226_5;
       "MDO".SPARE_226_6 := "PDO".SPARE_226_6;
       "MDO".SPARE_226_7 := "PDO".SPARE_226_7;
       "MDO".HOR_OPP_K8 := "PDO".HOR_OPP_K8;
       "MDO".LMP_RD_K8 := "PDO".LMP_RD_K8;
       "MDO".LMP_YE_K8 := "PDO".LMP_YE_K8;
       "MDO".LMP_GN_K8 := "PDO".LMP_GN_K8;
       "MDO".LMP_BU_K8 := "PDO".LMP_BU_K8;
       "MDO".XT_ROT_ENB := "PDO".XT_ROT_ENB;
       "MDO".XT_LFT_ENB := "PDO".XT_LFT_ENB;
       "MDO".XT_HDL_LFT_ENB := "PDO".XT_HDL_LFT_ENB;
       "MDO".XT_HDL_SW_ENB := "PDO".XT_HDL_SW_ENB;
       "MDO".FU_GCB_HDL_ON := "PDO".FU_GCB_HDL_ON;
       "MDO".LSR_SEN_PWR_ON := "PDO".LSR_SEN_PWR_ON;
       "MDO".SPARE_273_3 := "PDO".SPARE_273_3;
       "MDO".SPARE_273_4 := "PDO".SPARE_273_4;
       "MDO".SPARE_273_5 := "PDO".SPARE_273_5;
       "MDO".XT_HDL_SLID_FW := "PDO".XT_HDL_SLID_FW;
       "MDO".XT_HDL_SLID_BW := "PDO".XT_HDL_SLID_BW;
       "MDO".XT_CLP_TILT_BW := "PDO".XT_CLP_TILT_BW;
       "MDO".XT_CLP_TILT_FW := "PDO".XT_CLP_TILT_FW;
       "MDO".XT_CLP_TILT_BRK := "PDO".XT_CLP_TILT_BRK;
       "MDO".XT_CLP_ABV_OP := "PDO".XT_CLP_ABV_OP;
       "MDO".XT_CLP_ABV_CL := "PDO".XT_CLP_ABV_CL;
       "MDO".XT_CLP_ABV_BRK := "PDO".XT_CLP_ABV_BRK;
       "MDO".XT_CLP_ABV_RST := "PDO".XT_CLP_ABV_RST;
       "MDO".GCH_LFT_ENB := "PDO".GCH_LFT_ENB;
       "MDO".XT_CLP_BLW_OP := "PDO".XT_CLP_BLW_OP;
       "MDO".XT_CLP_BLW_CL := "PDO".XT_CLP_BLW_CL;
       "MDO".XT_CLP_BLW_BRK := "PDO".XT_CLP_BLW_BRK;
       "MDO".XT_CLP_BLW_RST := "PDO".XT_CLP_BLW_RST;
       "MDO".MCC_TEST_XT := "PDO".MCC_TEST_XT;
       "MDO".MCC_ENB_XT := "PDO".MCC_ENB_XT;
       "MDO".TCH_LFT_ENB := "PDO".TCH_LFT_ENB;
       "MDO".TCH_TILT_ENB := "PDO".TCH_TILT_ENB;
       "MDO".GTE_V_LFT_ENB := "PDO".GTE_V_LFT_ENB;
       "MDO".GTE_V_SW_ENB := "PDO".GTE_V_SW_ENB;
       "MDO".BEL_LFT_ENB := "PDO".BEL_LFT_ENB;
       "MDO".HOR_OPP_K9 := "PDO".HOR_OPP_K9;
       "MDO".LMP_RD_K9 := "PDO".LMP_RD_K9;
       "MDO".LMP_YE_K9 := "PDO".LMP_YE_K9;
       "MDO".LMP_GN_K9 := "PDO".LMP_GN_K9;
       "MDO".LMP_BU_K9 := "PDO".LMP_BU_K9;
END_FUNCTION_BLOCK

FUNCTION_BLOCK "PM_MAI"   // FB402, SCL
{ S7_Optimized_Access := 'FALSE' }
VERSION : 0.0
// --------------------------------------------------------------------------------
//     program:         PM_MAI
//     description :    automatically generated PM_MAI
//     name:            hp
//     date        :    03.02.2021
// 
//     revision:
//     name:
//     Date:
//                     (c)CGS
//     --------------------------------------------------------------------------------
   VAR
      y : Bool;
      count : Int := 8;
   END_VAR
   VAR_TEMP
      x : Bool;
   END_VAR
BEGIN


       "MAI".TRV_ACT_POS := "HAI".TRV_ACT_POS * 10.0;
       "MAI".TRV_ACT_POS_1 := "HAI".TRV_ACT_POS_1 * 10.0;
       "MAI".TRV_PRS_FIL_1 := "HAI".TRV_PRS_FIL_1 * 10.0;
       "MAI".TRV_PRS_FIL_2 := "HAI".TRV_PRS_FIL_2 * 10.0;
       "MAI".PYR_ACT_HTR_1_TMP := "HAI".PYR_ACT_HTR_1_TMP * 20.0;
       "MAI".ACT_PRS_AR_VSL := "HAI".ACT_PRS_AR_VSL * 20.0;
       "MAI".PYR_ACT_MELT_TMP := "HAI".PYR_ACT_MELT_TMP * 20.0;
       "MAI".GCH_PCR_ACT_PRS := "HAI".GCH_PCR_ACT_PRS * 10.0;
       "MAI".FCH_PCR_ACT_PRS := "HAI".FCH_PCR_ACT_PRS * 10.0;
       "MAI".FCH_BAR_ACT_PRS_100 := "HAI".FCH_BAR_ACT_PRS_100 * 10.0;
       "MAI".ACC_WTR_TMP := "HAI".ACC_WTR_TMP * 20.0;
       "MAI".ACC_WTR_PRS_IN := "HAI".ACC_WTR_PRS_IN * 20.0;
       "MAI".ACC_WTR_FLW_OUT := "HAI".ACC_WTR_FLW_OUT * 20.0;
       "MAI".ACC_WTR_FLW_IN := "HAI".ACC_WTR_FLW_IN * 20.0;
       "MAI".ACC_WTR_SPL_PRS := "HAI".ACC_WTR_SPL_PRS * 20.0;
       "MAI".ACC_SPARE_810 := "HAI".ACC_SPARE_810 * 20.0;
END_FUNCTION_BLOCK

FUNCTION_BLOCK "PM_MAO"   // FB403, SCL
{ S7_Optimized_Access := 'FALSE' }
VERSION : 0.0
// --------------------------------------------------------------------------------
//     program:         PM_MAO
//     description :    automatically generated PM_MAO
//     name:            hp
//     date        :    03.02.2021
// 
//     revision:
//     name:
//     Date:
//                     (c)CGS
//     --------------------------------------------------------------------------------
   VAR
      y : Bool;
      count : Int := 8;
   END_VAR
   VAR_TEMP
      x : Bool;
   END_VAR
BEGIN


       "MAO".TRV_SET_POS := "HAO".TRV_SET_POS * 10.0;
       "MAO".TRV_SET_POS_1 := "HAO".TRV_SET_POS_1 * 10.0;
END_FUNCTION_BLOCK

FUNCTION_BLOCK "PM_INI_DI"   // FB404, SCL
{ S7_Optimized_Access := 'FALSE' }
VERSION : 0.0
// --------------------------------------------------------------------------------
//     program:         PM_INI_DI
//     description :    automatically generated PM_INI_DI
//     name:            hp
//     date        :    03.02.2021
// 
//     revision:
//     name:
//     Date:
//                     (c)CGS
//     --------------------------------------------------------------------------------
   VAR
      y : Bool;
      count : Int := 8;
   END_VAR
   VAR_TEMP
      x : Bool;
   END_VAR
BEGIN


       "PDI".SPARE_144_2 := false;
       "PDI".SPARE_144_3 := false;
       "PDI".SPARE_144_4 := false;
       "PDI".SPARE_144_5 := false;
       "PDI".SPARE_144_6 := false;
       "PDI".SPARE_144_7 := false;
END_FUNCTION_BLOCK

FUNCTION_BLOCK "PM_INI_AI"   // FB405, SCL
{ S7_Optimized_Access := 'FALSE' }
VERSION : 0.0
// --------------------------------------------------------------------------------
//     program:         PM_INI_AI
//     description :    automatically generated PM_INI_AI
//     name:            hp
//     date        :    03.02.2021
// 
//     revision:
//     name:
//     Date:
//                     (c)CGS
//     --------------------------------------------------------------------------------
   VAR
      y : Bool;
      count : Int := 8;
   END_VAR
   VAR_TEMP
      x : Bool;
   END_VAR
BEGIN


       "PAI".SPARE_484 := 0.0;
       "PAI".SPARE_486 := 0.0;
       "PAI".SPARE_1538 := 0.0;
       "PAI".SPARE_1540 := 0.0;
       "PAI".SPARE_1542 := 0.0;
       "PAI".SPARE := 0.0;
END_FUNCTION_BLOCK

FUNCTION_BLOCK "BM_VAC_MAIN"   // FB500, SCL
{ S7_Optimized_Access := 'FALSE' }
VERSION : 0.0
// -----------------------------------------------------------------------------------
// program:             BM_VAC_MAIN
//     description :    Vacuum control
//     name:            hp
//     date        :    10.11.99
// 
//     revision    :    control sequence for motor control valve V1 for EKZ 2700 added       
//     name        :    G. Eibelsh鋟ser
//     Date        :    28.07.2000
//     
//     revision    :    delay time to open motor control valve after Pump P1 is on 
//                      EKZ 2700 added       
//     name        :    G. Eibelsh鋟ser
//     Date        :    28.07.2000
// 
//     
// 
//     
//                     (c)CGS
// -----------------------------------------------------------------------------------
   VAR
      P1_DATA : Array[1..8] of Byte;
      V1_OPEN_REQ : Bool;
      V1_CLOSE_REQ : Bool;
      P1_IS_ON : Bool;
      P3_IS_ON : Bool;
      V2_ONDELAY_OVER : Bool;
      V3_ONDELAY_OVER : Bool;
      P1_NOT_READY : Bool;
      P2_NOT_READY : Bool;
      P3_NOT_READY : Bool;
      Flt_P1 : Bool;
      Flt_P2 : Bool;
      Flt_P3 : Bool;
      PRS_FDR_FNC_OK : Bool;
      mob_fdr_p3_on_req : Bool;
      mob_fdr_p3_off_req : Bool;
      mob_fdr_v24_cl_req : Bool;
      mob_fdr_v24_opn_req : Bool;
      mob_fdr_v3_2_cl_req : Bool;
      mob_fdr_v3_2_opn_req : Bool;
      v5_auto_cl_req : Bool;
      v5_auto_opn_req : Bool;
      v6_auto_opn_req : Bool;
      v6_auto_cl_req : Bool;
      v6_cl_dly_run : Bool;
      v6_auto_cl_req_dly : Bool;
      cgt_v_cld_prv : Bool;
      V9_2_dly_op : Bool;
      V9_2_dly_cl : Bool;
      V9_1_dly_op : Bool;
      V9_1_dly_cl : Bool;
      BI_TMR_APS_FCH : Word;   // internal time values
      BI_TMR_APS_GCH : Word;
      BI_TMR_APS_FDR : Word;
      BI_TMR_APS_FIL : Word;
      BI_TMR_APS_BY_FIL : Word;
      BI_TMR_V1_ONDEL : Word;
      BI_TMR_V2_ONDEL : Word;
      BI_TMR_V3_ONDEL : Word;
      BI_TMR_P1_ONDEL : Word;
      BI_TMR_P3_ONDEL : Word;
      FltTimeV2_1 : Int;
      FltTimeV2_11 : Int;
      FltTimeV3 : Int;
      FltTimeV3_3 : Int;
      FltTimeV3_4 : Int;
      FltTimeV22_1 : Int;
      FltTimeV7 : Int;
      FltTimeP1 : Int;
      FltTimeP2 : Int;
      FltTimeP3 : Int;
      tmp_flt_p1_dly : Int;
      tmp_flt_p2_dly : Int;
      p1_on_dly : Int;
      p1_seal_gas_off_dly : Int;
      TimeV7_UP : Int;
      TimeV7_DN : Int;
      TimeV7_SW_IN : Int;
      TimeV7_SW_OUT : Int;
      i : Int;
      v21_not_open_dly : Int;
      DelayV9_1 : Int;
      DelayV9_2 : Int;
      onTimeV9_2 : Int;
      TRV_SET_POS : Real;   // position V1 (0...100 %)
      TRV_SET_POS_V1_1 : Real;
      TRV_POS_INC : Real;
   END_VAR
   VAR_TEMP
      iTime : S5Time;   // Return value function S_ODT (not used)
      Dprd_P1_RetVal : Int;
   END_VAR
   VAR CONSTANT
      DELAY_TIME_V1_ON : Time := T#30S;   // Delay open V1 after v2_1 on
      DELAY_TIME_V2_ON : Time := T#1M;   // Delay open V2_x after pump on
      DELAY_TIME_V3_ON : Time := T#1M;   // Delay open V3 after pump on
      DELAY_APS_FCH : Time := T#1S;   // Delay for APS furnace
      DELAY_APS_GCH : Time := T#1S;   // Delay for APS gate
      DELAY_APS_FDR : Time := T#3S;   // Delay for APS feeder
      DELAY_APS_FIL : Time := T#2S;   // Delay for APS main filter
      DELAY_APS_BY_FIL : Time := T#2S;   // Delay for APS bypass filter
      nc_bool : Bool := FALSE;   // not connected
      prs_hyst_ar_vsl : Real := 0.2;   // pressure hysteries argon tank in [bar]
   END_VAR
BEGIN

       //set alarm when compressed air pressure is low
       //---------------------------------------------
       "FLT".COMP_ACC_AIR_PRS_LOW    := NOT "PDI".COMP_AIR_OK;
       "FLT".COMP_SPL_AIR_PRS_LOW    := NOT "PDI".COMP_AIR_2_OK;

       //----------------------------------------------------------------------
       // Calculate pressure values
       //----------------------------------------------------------------------

       // furnace
       //--------
       IF ("PAI".FCH_PCR_ACT_PRS< 95.0) AND ("PAI".FCH_PCR_ACT_PRS>5.0) AND ("PAI".FCH_BAR_ACT_PRS_100>0.0) AND ("PAI".FCH_BAR_ACT_PRS_100<99.0)THEN
           "AV".ACT_PRS_FCH := "PAI".FCH_BAR_ACT_PRS_100;
       ELSE
           "AV".ACT_PRS_FCH := "PAI".FCH_PCR_ACT_PRS;
       END_IF;                                  
       "DIS".ACT_PRS_CLF := "AV".ACT_PRS_FCH;

       // gate
       //-----
       "AV".ACT_PRS_GCH := "PAI".GCH_PCR_ACT_PRS;
       "DIS".ACT_PRS_CGT := "AV".ACT_PRS_GCH;

       // feeder
       //-------
       IF "DV".MOB_FDR_V11_INST AND "DV".MOB_FDR_CON THEN
          "AV".ACT_PRS_FDR := "P_BM_FDR_PCR_ACT_PRS":P;
       ELSE
          "AV".ACT_PRS_FDR := 1000.0;
       END_IF;                                  
       "DIS".ACT_PRS_FDR := "AV".ACT_PRS_FDR;

       //calculate pressure difference feeder - furnace chamber 
       //------------------------------------------------------
       "AV".DIFF_PRS_FDR_FNC := "AV".ACT_PRS_FDR - "AV".ACT_PRS_FCH;

       IF (("AV".DIFF_PRS_FDR_FNC >= 0.0) AND ("AV".DIFF_PRS_FDR_FNC <= "CNF".MAX_DIFF_PRS_FDR_FNC))
       OR ("DV".APS_FDR_DELAYED AND "DV".APS_FCH_DELAYED)
       OR "PDI".LS_V11_OP                                THEN

           #PRS_FDR_FNC_OK := TRUE; 
       ELSE
           #PRS_FDR_FNC_OK := FALSE;
       END_IF;

